(* CODESYS project CtaAppAntrieb_2.0.0.1.library
   Description: Antriebs Library der CTA
   Version: 2.0.0.1
   Title: CtaAppAntrieb
   Author: SIS
   DocFormat: reStructuredText
   LanguageModelAttribute: qualified-access-only
   Placeholder: CtaAppAntrieb
   DefaultNamespace: CtaAppAntrieb
   CompiledLibraryCompatibilityVersion: CODESYS V3.5 SP20 Patch 5
   Company: CTA

Project tree, tasks and I/O mapping:
  libraries: Standard, 3.5.18.0 (System); CtaAppBasic, 1.0.0.0 (CTA); CtaAppBmk, 2.0.0.0 (CTA); CtaSysConfig, 2.0.0.0 (CTA); VisuDialogs, 3.5.16.20 (System); VisuSymbols, 4.5.0.0 (System); CtaSysMotor, 1.0.0.0 (CTA); CtaAppReport, 2.0.0.0 (CTA); CtaVisHelp, 1.0.0.0 (CTA); CtaVisSymbols, 2.0.0.0 (CTA); CtaAppDumper, 2.0.0.0 (CTA); CtaAppInfluxLog, 1.0.0.1 (CTA); CtaSysIO, 2.0.0.0 (CTA); CtaAppModbusSpezifikation, 1.0.0.1 (CTA); CtaVisApps, 1.0.0.0 (CTA); CtaVisUser, 1.0.0.0 (CTA)
  40 Visualizations/
    ICON/
      ANTRIEB_RIGHT/
        ANTRIEB_RIGHT_BELOW/
          visualisation VIS_ANTRIEB_RIGHT_BELOW
          visualisation VIS_ANTRIEB_RigthBelowCheckIsEnabled
          visualisation VIS_ANTRIEB_RigthBelowCheckQuerry
        ANTRIEB_RIGHT_ABOVE/
          visualisation VIS_ANTRIEB_RigthAboveCheckQuerry
          visualisation VIS_ANTRIEB_RIGHT_ABOVE
          visualisation VIS_ANTRIEB_RigthAboveCheckIsEnabled
      ANTRIEB_BASE/
        visualisation CommandOn
        visualisation ValueUpDwn
        ICON/
          visualisation Icon_Left
          visualisation Icon_Right
        visualisation ValueDwnUp
      ANTRIEB_LEFT/
        ANTRIEB_LEFT_BELOW/
          visualisation VIS_ANTRIEB_LEFT_BELOW
          visualisation VIS_ANTRIEB_LeftBelowCheckIsEnabled
          visualisation VIS_ANTRIEB_LeftBelowCheckQuerry
        ANTRIEB_LEFT_ABOVE/
          visualisation VIS_ANTRIEB_LEFT_ABOVE
          visualisation VIS_ANTRIEB_LeftAboveCheckIsEnabled
          visualisation VIS_ANTRIEB_LeftAboveCheckQuerry
    POPUP/
      visualisation POPUP_ANTRIEB
      PARAMETER/
        visualisation VIS_ANTRIEB_PARAMETER
        visualisation VIS_ANTRIEB_PARAMETER_LISTE
        AT_ParameterBase/
          visualisation VIS_ANTRIEB_PARAMETER_BASE0
          visualisation VIS_ANTRIEB_PARAMETER_BASE
        AT_Data/
          visualisation VIS_ANTRIEB_PARAMETER_DATA0
          visualisation VIS_ANTRIEB_PARAMETER_DATA
        AT_Fuse/
          visualisation VIS_ANTRIEB_PARAMETER_FUSES0
          visualisation VIS_ANTRIEB_PARAMETER_FUSES
        AT_IO/
          visualisation VIS_ANTRIEB_PARAMETER_IO0
          visualisation VIS_ANTRIEB_PARAMETER_IO1
          visualisation VIS_ANTRIEB_PARAMETER_IO
          visualisation VIS_ANTRIEB_PARAMETER_IO2
          visualisation VIS_ANTRIEB_PARAMETER_IO3
          visualisation VIS_ANTRIEB_PARAMETER_IO4
        AT_InfluxDb/
          visualisation VIS_ANTRIEB_PARAMETER_TRENDLOG
          visualisation VIS_ANTRIEB_PARAMETER_TRENDLOG0
        visualisation VIS_ANTRIEB_POPUP_IO_ITF
      visualisation VIS_ANTRIEB_LISTE
      MANUAL/
        visualisation VIS_ANTRIEB_MANUAL
      OVERVIEW/
        visualisation VIS_ANTRIEB_OVERVIEW
      BUS/
        visualisation AT_BUS
        visualisation AT_BUS_SW0_Detail
        visualisation AT_BUS_CW0_Detail
        visualisation AT_BUS_CS
        visualisation AT_BUS_SW1_Detail
        visualisation AT_BUS_SW2_Detail
      REPORTS/
        visualisation VIS_ANTRIEB_REPORTS
      IO/
        visualisation VIS_ANTRIEB_IO0
        visualisation VIS_ANTRIEB_IO
        visualisation VIS_ANTRIEB_IO1
  30 Program Organization Units/
    function block fbAntrieb [ST]: proHandOn, proAuto, proHandOff, proHandOnY, proHardWareHandModulAktive, actConfig, proConfigError, proIconNr, P_scBase_fbrYMax, P_scBase_fbrYMin, P_scBase_fbtLeadTime, P_scBase_fbtRunAfterTime, P_scBase_fbxControllMb, P_scBase_fbxEnable, P_scBase_fbxRegulatet, P_scData_fbudiOperatingHours, P_scData_fbudiOperationStarts, P_scFuse_fbxDoesAlarm, P_scFuse_fbxEnable, P_scFuse_fbxInputMb, P_scInfluxDb_fbxEnable, P_scIO_IsHand_fbxEnable, P_scIO_IsHand_fbxInputMb, P_scIO_IsNoError_fbiMaxErrorRetryAllowed, P_scIO_IsNoError_fbiTypeOfAck, P_scIO_IsNoError_fbtDelayRun, P_scIO_IsNoError_fbtDelayStartSps, P_scIO_IsNoError_fbxDoesAlarm, P_scIO_IsNoError_fbxEnable, P_scIO_IsNoError_fbxInputMb, P_scIO_IsOn_fbiMaxErrorRetryAllowed, P_scIO_IsOn_fbiTypeOfAck, P_scIO_IsOn_fbtDelayRun, P_scIO_IsOn_fbtDelayStart, P_scIO_IsOn_fbxDoesAlarm, P_scIO_IsOn_fbxEnable, P_scIO_IsOn_fbxInputMb, P_scIO_IsReady_fbxEnable, P_scIO_IsReady_fbxInputMb, P_scIO_IsValue_fbiMaxErrorRetryAllowed, P_scIO_IsValue_fbiTypeOfAck, P_scIO_IsValue_fbrMaxDiff, P_scIO_IsValue_fbtDelayRun, P_scIO_IsValue_fbtDelayStart, P_scIO_IsValue_fbxDoesAlarm, P_scIO_IsValue_fbxEnable, P_scIO_IsValue_fbxInputMb, P_scIO_RevisionSwitch_fbxEnable, P_scIO_RevisionSwitch_fbxInputMb, P_scManual_fbrManualOnY, P_scManual_fbuiManualState, P_scManual_fbxAlowManualOn, P_scMotorFuse_fbxDoesAlarm, P_scMotorFuse_fbxEnable, P_scMotorFuse_fbxInputMb, proRefToRonYDumper, actMbControll, actMbState, proModbusTest, proModbusStateWord, proModbusControllWord, proIsOn, proIsError, proIsWarning, proIsRegulatet, proIsEnabled, actState, proMotorIsOn, proIsHandOnOrOff, proIsReady, proLeadTime, proRunAfterTime, proIsOnY, proLeadTimeAktive, proRunAfterTimeAktive, proRevisionSwitchOk, proCountedHours, proCountedStarts, proStateSymbol, proCountedError, proCountedInfo, proCountedWarning, proITF_REPORTMANAGER, proGetDI_IsOn, metDI_IsOn, proNotShowDI_IsOn, proIsOn_ITF, metDI_RevisionSwitchOk, proNotShowDI_RevisionSwitchOk, proGetDI_RevisionSwitchOK, proRevisionSwitch_ITF, metDI_NoError, proNotShowDI_NoError, proGetDI_NoError, proNoError_ITF, proGetDI_FuseOK, metDI_ITF_FuseOK, proNotShowDI_FuseOk, proFuse_ITF, metDI_ITF_MotorHand, proNotShowDI_MotorHand, proGetDI_MotorHand, proHandModul_ITF, metDI_IsReady, proNotShowDI_Ready, proGetDI_IsReady, proReady_ITF, metDI_MotorFuseOk, proNotShowDI_MotorFuseOk, proGetDI_MotorFuseOk, proMotorFuse_ITF, metDO_On, proOn_ITF, metAO_OnY, proOnY_ITF, proNotShowAI_ActualValue, metAI_ActualValue, proGetAI_ActualValue, proActualValue_ITF, proOnY, proOn, actVorlaufNachlauf, actPrioOfControll, actResetOnDisable, proEn, proEnSymbol, actTrendLog, actReport, proLockDown, proAvailable, proAcknowlege
    function fcGetBigerStringValue [ST]
    function fcCheckQuerryAndIconReturn [ST]
  00000000-0000-0000-0000-000000000000|D:\CoDeSys\LibrariesV3\trunk\Intern\CAA\CAA Template\3.4.0.0 draft\Placeholder.xml
  00000000-0000-0000-0000-000000000000|D:\CoDeSys\LibrariesV3\trunk\Intern\CAA\CAA Template\3.2.0.3 draft\Prefix.pdf
  00000000-0000-0000-0000-000000000000|D:\CoDeSys\LibrariesV3\trunk\Intern\CAA\CAA Template\3.5.2.0 draft\Placeholder.xml
  20 Structs/
    data type scParameter
    IO/
      data type scIO_IsOn
      data type scIO_IsNoError
      data type scIO_IsReady
      data type scIO_RevisionSwitch
      data type scIO_IsValue
      data type scIO_IsHand
    BASE/
      data type scBase
    DATA/
      data type scData
    FUSE/
      data type scFuse
      data type scMotorFuse
    InfluxDb/
      data type scInfluxDb
    MANUAL/
      data type scManual
  50 Images/
  10 Documenation/
    global variables VersionHistory
    global variables readMe
  21 Interface/
    interface ITF_ANTRIEB: proModbusTest, proModbusStateWord, proModbusControllWord, proConfigError, P_scIO_IsHand_fbxEnable, P_scIO_IsHand_fbxInputMb, P_scIO_IsNoError_fbxEnable, P_scIO_IsNoError_fbxInputMb, P_scIO_IsNoError_fbxDoesAlarm, P_scIO_IsNoError_fbtDelayStartSps, P_scIO_IsNoError_fbtDelayRun, P_scIO_IsNoError_fbiTypeOfAck, P_scIO_IsNoError_fbiMaxErrorRetryAllowed, P_scIO_IsOn_fbxInputMb, P_scIO_IsOn_fbxEnable, P_scIO_IsOn_fbtDelayStart, P_scIO_IsOn_fbxDoesAlarm, P_scIO_IsOn_fbtDelayRun, P_scIO_IsOn_fbiTypeOfAck, P_scIO_IsOn_fbiMaxErrorRetryAllowed, P_scIO_IsReady_fbxEnable, P_scIO_IsReady_fbxInputMb, P_scIO_IsValue_fbxInputMb, P_scIO_IsValue_fbxEnable, P_scIO_IsValue_fbxDoesAlarm, P_scIO_IsValue_fbtDelayStart, P_scIO_IsValue_fbtDelayRun, P_scIO_IsValue_fbiTypeOfAck, P_scIO_IsValue_fbiMaxErrorRetryAllowed, P_scIO_IsValue_fbrMaxDiff, P_scIO_RevisionSwitch_fbxEnable, P_scIO_RevisionSwitch_fbxInputMb, P_scBase_fbxEnable, P_scBase_fbxRegulatet, P_scBase_fbxControllMb, P_scBase_fbrYMin, P_scBase_fbrYMax, P_scBase_fbtLeadTime, P_scBase_fbtRunAfterTime, P_scFuse_fbxEnable, P_scFuse_fbxInputMb, P_scFuse_fbxDoesAlarm, P_scMotorFuse_fbxInputMb, P_scMotorFuse_fbxEnable, P_scMotorFuse_fbxDoesAlarm, P_scManual_fbxAlowManualOn, P_scManual_fbuiManualState, P_scManual_fbrManualOnY, P_scInfluxDb_fbxEnable, P_scData_fbudiOperationStarts, P_scData_fbudiOperatingHours, proRefToRonYDumper, proCountedError, proCountedInfo, proITF_REPORTMANAGER, proCountedWarning, proCountedHours, proCountedStarts, proGetDI_MotorHand, proNotShowDI_MotorHand, proHandModul_ITF, proNotShowAI_ActualValue, proGetAI_ActualValue, proActualValue_ITF, proNotShowDI_NoError, proGetDI_NoError, proNoError_ITF, proNotShowDI_RevisionSwitchOk, proGetDI_RevisionSwitchOK, proRevisionSwitch_ITF, proNotShowDI_IsOn, proGetDI_IsOn, proIsOn_ITF, proNotShowDI_MotorFuseOk, proGetDI_MotorFuseOk, proMotorFuse_ITF, proNotShowDI_FuseOk, proGetDI_FuseOK, proFuse_ITF, proNotShowDI_Ready, proGetDI_IsReady, proReady_ITF, proOn_ITF, proOnY_ITF, proIsRegulatet, proIsHandOnOrOff, proRunAfterTimeAktive, proLeadTimeAktive, proIsReady, proAuto, proHandOn, proIsError, proIsWarning, proEn, proHardWareHandModulAktive, proIsEnabled, proMotorIsOn, proHandOff, proRevisionSwitchOk, proHandOnY, proEnSymbol, proIsOn, proIsOnY, proLeadTime, proOn, proOnY, proRunAfterTime, proStateSymbol, proLockDown, proAvailable, proAcknowlege, proIconNr
  11 Library Parameter/
  12 Konstanten/
    global variables GlobalKonstant
  60 Textlisten/
    text list GlobalTextList
    text list Error
    text list Info
    text list Warnung
  13 Globale Variablen/
  5ce3da45-db07-42e7-a21c-a00fff4ed8f6|C:\Users\sis\Downloads\dip-switch.svg
  5ce3da45-db07-42e7-a21c-a00fff4ed8f6|C:\Users\sis\Downloads\lightning-bolt-circle.svg
  5ce3da45-db07-42e7-a21c-a00fff4ed8f6|C:\Users\sis\Downloads\sine-wave.svg
  5ce3da45-db07-42e7-a21c-a00fff4ed8f6|C:\Users\sis\Downloads\eye.svg
  5ce3da45-db07-42e7-a21c-a00fff4ed8f6|C:\Users\sis\Downloads\lan.svg
*)

// 20 Structs/scParameter
{attribute 'pack_mode' := '1'} 
TYPE scParameter :
    STRUCT
		
        scBase              :   scBase;					// Basisparameter		
        scFuse              :   scFuse;					// Parameter Sicherung
        scMotorFuse         :   scMotorFuse;			// Parameter Motorsicherung
        scIO_RevisionSwitch :   scIO_RevisionSwitch;	// Parameter Revisionsschalter 
        scIO_IsReady        :   scIO_IsReady;   		// Parameter Bereitmeldung
        scIO_IsOn           :   scIO_IsOn;				// Parameter Betriebsrückmeldung
        scIO_IsNoError      :   scIO_IsNoError;			// Parameter Störmeldung
        scIO_IsValue        :   scIO_IsValue;			// Parameter Istwert
        scIO_IsHand         :   scIO_IsHand;        	// Parameter Handwert
        scManual            :   scManual;				// Parameter Handbedienung
        scData              :   scData;					// Parameter Betriebsdaten 
        scInfluxDb          :   scInfluxDb;				// Parameter Datenbankaufzeichung
    END_STRUCT
END_TYPE

// 20 Structs/IO/scIO_IsOn
{attribute 'pack_mode' := '1'} 
TYPE scIO_IsOn :
    STRUCT
        fbxEnable                    : CtaSysConfig.fbBOOL;	// Betriebsrückmeldung wird ausgewertet
        fbxInputMb                   : CtaSysConfig.fbBOOL; // Betriebsrückmeldung via Modbus  
        fbxDoesAlarm                 : CtaSysConfig.fbBOOL; // Ausstehende Betriebsrückmeldung löst Fehler aus 
        fbtDelayStart                : CtaSysConfig.fbTIME; // Verzögerung für Srörungsausgabe
        fbtDelayRun                  : CtaSysConfig.fbTIME; // Verzögerung für Störungsausgabe während Betrieb 
        fbiTypeOfAck               	 : CtaSysConfig.fbINT;  // Art der FehlerQuittierung 0 = Automatisch, 1 = Quittierpflichtig, 2 = Selbstquittierend bis N  
        fbiMaxErrorRetryAllowed      : CtaSysConfig.fbINT;  // Anzahl möglicher Selbstquittierungen    
    END_STRUCT
END_TYPE

// 20 Structs/IO/scIO_IsNoError
{attribute 'pack_mode' := '1'} 
TYPE scIO_IsNoError :
    STRUCT
        fbxEnable                    : CtaSysConfig.fbBOOL;	// Störkontakt wird ausgewertet
        fbxInputMb                   : CtaSysConfig.fbBOOL; // Störkontaktstatus via Modbus
        fbxDoesAlarm                 : CtaSysConfig.fbBOOL;	// Störung löst Fehler aus
        fbtDelayStartSps             : CtaSysConfig.fbTIME; // Verzögerung für Srörungsausgabe
        fbtDelayRun                  : CtaSysConfig.fbTIME; // Verzögerung für Störungsausgabe während Betrieb 
        fbiTypeOfAck               	 : CtaSysConfig.fbINT;	// Art der FehlerQuittierung 0 = Automatisch, 1 = Quittierpflichtig, 2 = Selbstquittierend bis N 
        fbiMaxErrorRetryAllowed      : CtaSysConfig.fbINT;	// Anzahl möglicher Selbstquittierungen
    END_STRUCT
END_TYPE

// 20 Structs/IO/scIO_IsReady
{attribute 'pack_mode' := '1'} 
TYPE scIO_IsReady :
    STRUCT
        fbxEnable                    : CtaSysConfig.fbBOOL;	// Bereitmeldung wird ausgewertet 
        fbxInputMb                   : CtaSysConfig.fbBOOL; // Bereitmeldung üver Modbus         
    END_STRUCT
END_TYPE

// 20 Structs/IO/scIO_RevisionSwitch
{attribute 'pack_mode' := '1'} 
TYPE scIO_RevisionSwitch :
    STRUCT
        fbxEnable                   : CtaSysConfig.fbBOOL;	// Revisionsschalter wird ausgewertet
        fbxInputMb                  : CtaSysConfig.fbBOOL;	// Revisionsschalterstatus via Modbus
    END_STRUCT
END_TYPE

// 20 Structs/IO/scIO_IsValue
{attribute 'pack_mode' := '1'} 
TYPE scIO_IsValue :
    STRUCT
        fbxEnable                    : CtaSysConfig.fbBOOL;	// Iststellwert wird ausgewertet
        fbxInputMb                   : CtaSysConfig.fbBOOL; // Iststellwert via Modbus    
        fbxDoesAlarm                 : CtaSysConfig.fbBOOL; // Zugrosse Abweichung löst Fehler aus  
        fbrMaxDiff                   : CtaSysConfig.fbREAL; // Maximal zulässige abweichung von Soll- zu Iststellwert
        fbtDelayStart                : CtaSysConfig.fbTIME; // Verzögerung für Srörungsausgabe
        fbtDelayRun                  : CtaSysConfig.fbTIME; // Verzögerung für Störungsausgabe während Betrieb 
		fbiTypeOfAck				 : CtaSysConfig.fbINT;  // Art der FehlerQuittierung 0 = Automatisch, 1 = Quittierpflichtig, 2 = Selbstquittierend bis N  
		fbiMaxErrorRetryAllowed		 : CtaSysConfig.fbINT;  // Anzahl möglicher Selbstquittierungen            
    END_STRUCT
END_TYPE

// 20 Structs/IO/scIO_IsHand
{attribute 'pack_mode' := '1'} 
TYPE scIO_IsHand :
    STRUCT
        fbxEnable                   : CtaSysConfig.fbBOOL;	// Handmodul wird ausgewertet
        fbxInputMb                  : CtaSysConfig.fbBOOL;	// Handmodulstatus via Modbus
    END_STRUCT
END_TYPE

// 20 Structs/BASE/scBase
{attribute 'pack_mode' := '1'} 
TYPE scBase :
    STRUCT
        fbxEnable       :   CtaSysConfig.fbBOOL;	// Antriebsbaustein wird abgearbeitet
        fbxRegulatet    :   CtaSysConfig.fbBOOL;	// Antriebsstellwert wird geregelt
        fbxControllMb   :   CtaSysConfig.fbBOOL;	// Antriebsansteuerung erfolgt über Modbus
        fbrYMin         :   CtaSysConfig.fbREAL;	// Minimalstellwert des Antriebes
        fbrYMax         :   CtaSysConfig.fbREAL;	// Maximalstellwert des Antriebes
        fbtLeadTime     :   CtaSysConfig.fbTIME;	// Vorlaufzeit des Antriebs
        fbtRunAfterTime :   CtaSysConfig.fbTIME;	// Nachlaufzeit des Antriebs
    END_STRUCT
END_TYPE

// 20 Structs/DATA/scData
{attribute 'pack_mode' := '1'} 
TYPE scData :
    STRUCT
        fbudiOperationStarts    :   CtaSysConfig.fbUDINT;	// Anzahl Einschaltungen des Antriebs
        fbudiOperatingHours     :   CtaSysConfig.fbUDINT;	// Anzahl Betriebsstunden des Antriebs
    END_STRUCT
END_TYPE

// 20 Structs/FUSE/scFuse
{attribute 'pack_mode' := '1'} 
TYPE scFuse :
    STRUCT
        fbxEnable               : CtaSysConfig.fbBOOL;	// Sicherung ist vorhanden
        fbxInputMb              : CtaSysConfig.fbBOOL;	// Sicherungsstatus via Modbus
        fbxDoesAlarm            : CtaSysConfig.fbBOOL;	// Defekte Sicherung löst Fehler aus
    END_STRUCT
END_TYPE

// 20 Structs/FUSE/scMotorFuse
{attribute 'pack_mode' := '1'} 
TYPE scMotorFuse :
    STRUCT
        fbxEnable             : CtaSysConfig.fbBOOL;	// Sicherung ist vorhanden
        fbxInputMb            : CtaSysConfig.fbBOOL;    // Sicherungsstatus via Modbus
        fbxDoesAlarm          : CtaSysConfig.fbBOOL;    // Defekte Sicherung löst Fehler aus  
    END_STRUCT
END_TYPE

// 20 Structs/InfluxDb/scInfluxDb
{attribute 'pack_mode' := '1'} 
TYPE scInfluxDb :
    STRUCT
        fbxEnable       :   CtaSysConfig.fbBOOL;	// Aktivierung der Trendaufzeichnung
    END_STRUCT
END_TYPE

// 20 Structs/MANUAL/scManual
{attribute 'pack_mode' := '1'} 
TYPE scManual :
    STRUCT
        fbxAlowManualOn         : CtaSysConfig.fbBOOL; 	// Manuelle ansteuerung des Antriebs zulässig   
        fbuiManualState         : CtaSysConfig.fbUINT;	// 0 = Auto ; 1 = Manual Off 2 = Manual On
        fbrManualOnY            : CtaSysConfig.fbREAL; 	// Manueller Stellwert für Antrieb
    END_STRUCT
END_TYPE

// 10 Documenation/VersionHistory
(* 

.. image:: ../../Images/CTA_Logo.jpg
   :align: right
   :width: 15% 

**Vorlage**   


============ =========== =========== ============================================
**Date**     **Version** **Author**  **Change**
------------ ----------- ----------- --------------------------------------------
04.03.2021   0.0.0.0     SIS         Vorlage erstellt

============ =========== =========== ============================================


*)
VAR_GLOBAL
    stInfo : STRING:= '0.0.0.0, Vorlage, CTA';
END_VAR

// 10 Documenation/readMe

(*

**ReadMe**
 
|	**Empfehlung**
|
|	Die Bibliothek CtaAppAntrieb wurde universal gestaltet, dadurch können verschiedene Komponenten damit angesteuert werden.
|	Instanzieren Sie den CtaAppAntrieb.fbAntrieb in ihrem Funktionsbaustein oder POU beispielsweise als fbPumpeX oder fbVentiX abhängig der Komponente. (X = Nr.) 
|	Deklarieren Sie die Struktur Variable welche als Parameter und zur ansteuerung dienen wie im Code beispiel.
|  
| *Beispiel* 

+-----------------------+---------------------------------------------------------------------------------------------------------------------------------------------------------------------------------------------------------------------------------------------------------------------------------------------------------------------------------------------------------------------------------------------------------------------------------------+
| Beschreibung          |  Code                                                                                                                                                                                                                                                                                                                                                                                                                                 |
+=======================+=======================================================================================================================================================================================================================================================================================================================================================================================================================================+
| Pou oder SmFb         | .. code-block:: codesys                                                                                                                                                                                                                                                                                                                                                                                                               |
|                       |                                                                                                                                                                                                                                                                                                                                                                                                                                       |
|                       |	// Deklaration als VAR im POU oder dem selbsterstellten Funktionsbaustein                                                                                                                                                                                                                                                                                                                                                       	|
|                       |   VAR   																																																																																																								|
|						|	    (*Pumpe1*)																																																		 																																																				|
|						|		fbPumpe1			: CtaAppAntrieb.fbAntrieb;                                                                                                                                                                                                                                                                                                                                                              					|
|                       | 		(*Ventilator1*)																																																																																																					|
| 						|		fbVenti1			: CtaAppAntrieb.fbAntrieb;																																																																																													|
| 						|	END_VAR                                                                                                                                                                                                                                                                                                                                                                                                                         	|
+-----------------------+---------------------------------------------------------------------------------------------------------------------------------------------------------------------------------------------------------------------------------------------------------------------------------------------------------------------------------------------------------------------------------------------------------------------------------------+
| Code für Init         | .. code-block:: codesys                                                                                                                                                                                                                                                                                                                                                                                                               |
|                       |   																																																																																																									|
| 						|	// Kopieren des nachfolgenden Codes in eine Action zur Initialisierung der Parameter. Zum Beispiel actConfig.																																																																														|
|                       |	{region "Parameter Pumpe1"}                                                                                                                                                                                                                                                                                                                                                                                                     	|
| 						|		(*Basis*)																																																																																																						|
|						|		fbPumpe1.scParameter.scBase.fbxEnable               		(_wertInit :=  TRUE																			);		//P1 Ein- Ausschalten des Antriebs																																																								|
|						|		fbPumpe1.scParameter.scBase.fbxRegulatet					(_wertInit :=  TRUE																			);		//P2 Antrieb ist geregelt / nicht geregelt																																																						| 
|						|		fbPumpe1.scParameter.scBase.fbxControllMb					(_wertInit := FALSE																			);		//P3 Ansteuerung oder Signalauswertung über Modbus																																																				| 
|						|		fbPumpe1.scParameter.scBase.fbrYMin							(_wertInit :=   0.0									, _minInit :=   0.0, _maxInit := 100.0	);		//P4 Minimaler Stellwert des Antriebs																																																							| 
|						|		fbPumpe1.scParameter.scBase.fbrYMax							(_wertInit := 100.0									, _minInit :=   0.0, _maxInit := 100.0	);		//P5 Maximaler Stellwert des Antriebs																																																							|
|						|		fbPumpe1.scParameter.scBase.fbtLeadTime						(_wertInit := T#30S									, _minInit :=      , _maxInit :=		);		//P6 Vorlaufzeit des Antriebs																																																									| 
|						|		fbPumpe1.scParameter.scBase.fbtRunAfterTime					(_wertInit := T#60S									, _minInit :=	   , _maxinit :=		);		//P7 Nachlaufzeit des Antriebs																																																									| 
|						|		(*Sicherungen*)																																																		 																																																			| 
|						|		fbPumpe1.scParameter.scFuse.fbxEnable						(_wertInit := FALSE																			);		//P8 Sicherung ist vorhanden / nicht vorhanden																	    																																			| 
|						|		fbPumpe1.scParameter.scFuse.fbxInputMb						(_wertInit := FALSE																			);		//P9 Ansteuerung oder Signalauswertung über Modbus																												    																							| 
|						|		fbPumpe1.scParameter.scFuse.fbxDoesAlarm					(_wertInit := FALSE																			);		//P10 Abfallendes Signal löst Fehler aus																											    																										| 
|						|		(*Motorsicherung*)																																																											 																																	  								| 
|						|		fbPumpe1.scParameter.scMotorFuse.fbxEnable					(_wertInit := FALSE																			);		//P11 Leistungsschutzschalter ist vorhanden / nicht vorhanden																    																																| 
|						|		fbPumpe1.scParameter.scMotorFuse.fbxInputMb					(_wertInit := FALSE																			);		//P12 Ansteuerung oder Signalauswertung über Modbus																																								   	 											| 
|						|		fbPumpe1.scParameter.scMotorFuse.fbxDoesAlarm				(_wertInit := FALSE																			);		//P13 Abfallendes Signal löst Fehler aus																														    																							| 
|						|		(*Revisionsschalter*)																																																											 																																							    | 
|						|		fbPumpe1.scParameter.scIO_RevisionSwitch.fbxEnable			(_wertInit := FALSE																			);		//P14 Revisionsschalter ist vorhanden / nicht vorhanden																																				    														| 
|						|		fbPumpe1.scParameter.scIO_RevisionSwitch.fbxInputMb			(_wertInit := FALSE																			);		//P15 Ansteuerung oder Signalauswertung über Modbus																																		    																	| 
|						|		(*Ready- Input*)																																																																																																			    | 
|						|		fbPumpe1.scParameter.scIO_IsReady.fbxEnable					(_wertInit := FALSE																			);		//P16 Readysignal ist vorhanden / nicht vorhanden																																	    																		| 
|						|		fbPumpe1.scParameter.scIO_IsReady.fbxInputMb				(_wertInit := FALSE																			);		//P17 Ansteuerung oder Signalauswertung über Modbus																																										    									| 
|						|		(*Betriebsrückmeldung*)																																																										 																																								    | 
|						|		fbPumpe1.scParameter.scIO_IsOn.fbxEnable					(_wertInit := FALSE																			);		//P18 Betriebsrückmeldung ist vorhanden / nicht vorhanden																														   																				| 
|						|		fbPumpe1.scParameter.scIO_IsOn.fbxInputMb					(_wertInit := FALSE																			);		//P19 Ansteuerung oder Signalauswertung über Modbus																																								    											| 
|						|		fbPumpe1.scParameter.scIO_IsOn.fbxDoesAlarm					(_wertInit := FALSE																			);		//P20 Fehlendes oder abfallendes Signal löst Fehler aus				   																																															| 
|						|		fbPumpe1.scParameter.scIO_IsOn.fbtDelayStart				(_wertInit := T#00S									, _minInit :=      , _maxInit :=  		);		//P21 Verzögerung der Fehlerausgabe nach Start																						   																															| 
|						|		fbPumpe1.scParameter.scIO_IsOn.fbtDelayRun					(_wertInit := T#00S									, _minInit :=      , _maxInit :=  		);		//P22 Verzögerung der Fehlerausgabe während Betrieb															    																																				| 
|						|		fbPumpe1.scParameter.scIO_IsOn.fbiTypeOfAck					(_wertInit :=     1									, _minInit :=     0, _maxInit :=    2	);		//P23 Art der Quittierung des Fehlers (auto, quittierend, quittierend bid n Meldung																																												|
|						|		fbPumpe1.scParameter.scIO_IsOn.fbiMaxErrorRetryAllowed		(_wertInit :=     3									, _minInit :=     0, _maxInit :=    5	);		//P24 Maximale Anzahl Wiederholungen bis zur Sperrung der Anlage																																																|
|						|		(*Fehler- Input*)																																																																																																			    | 
|						|		fbPumpe1.scParameter.scIO_IsNoError.fbxEnable				(_wertInit := FALSE																			);		//P25 Fehlerinput ist vorhanden / nicht vorhanden																																		    																	| 
|						|		fbPumpe1.scParameter.scIO_IsNoError.fbxInputMb				(_wertInit := FALSE																			);		//P26 Ansteuerung oder Signalauswertung über Modbus																																																			    | 
|						|		fbPumpe1.scParameter.scIO_IsNoError.fbxDoesAlarm			(_wertInit := FALSE																			);		//P27 Fehlendes oder abfallendes Signal löst Fehler aus				   																																														    | 
|						|		fbPumpe1.scParameter.scIO_IsNoError.fbtDelayStartSps		(_wertInit := T#00S									, _minInit :=      , _maxInit :=  		);		//P28 Verzögerung der Fehlerausgabe nach Start																																																			    	| 
|						|		fbPumpe1.scParameter.scIO_IsNoError.fbtDelayRun				(_wertInit := T#00S									, _minInit :=      , _maxInit :=  		);		//P29 Verzögerung der Fehlerausgabe während Betrieb																																																			    | 
|						|		fbPumpe1.scParameter.scIO_IsNoError.fbiTypeOfAck			(_wertInit :=     1 								, _minInit :=     0, _maxInit :=    2	);		//P30 Art der Quittierung des Fehlers (auto, quittierend, quittierend bid n Meldung																																										    	| 
|						|		fbPumpe1.scParameter.scIO_IsNoError.fbiMaxErrorRetryAllowed	(_wertInit :=     3 								, _minInit :=     0, _maxInit :=    5	);		//P31 Maximale Anzahl Wiederholungen bis zur Sperrung der Anlage																																										    					| 
|						|		(*Ist - Wert*)																																																																																																				    | 
|						|		fbPumpe1.scParameter.scIO_IsValue.fbxEnable					(_wertInit := FALSE																			);		//P32 Rückmeldung des Istwerts ist vorhanden / nicht vorhanden																																																	| 
|						|		fbPumpe1.scParameter.scIO_IsValue.fbxInputMb				(_wertInit := FALSE																			);		//P33 Ansteuerung oder Signalauswertung über Modbus																																																				| 
|						|		fbPumpe1.scParameter.scIO_IsValue.fbxDoesAlarm				(_wertInit := FALSE																			);		//P34 Unter oder überschreitung der Maximal erlaubten Differenz löst Fehler aus				   																																									| 
|						|		fbPumpe1.scParameter.scIO_IsValue.fbrMaxDiff				(_wertInit :=   0.0									, _minInit :=      , _maxInit :=		);		//P34 Maximal erlaubte Differenz des Stell- zum Istwert  			   																																															| 
|						|		fbPumpe1.scParameter.scIO_IsValue.fbtDelayStart				(_wertInit := T#00S									, _minInit :=      , _maxInit :=    	);		//P36 Verzögerung der Fehlerausgabe nach Start																																																					| 
|						|		fbPumpe1.scParameter.scIO_IsValue.fbtDelayRun				(_wertInit := T#00S									, _minInit :=      , _maxInit :=    	);		//P37 Verzögerung der Fehlerausgabe während Betrieb																																																				| 
|						|		fbPumpe1.scParameter.scIO_IsValue.fbiTypeOfAck				(_wertInit :=     1									, _minInit :=     0, _maxInit :=    2	);		//P38 Art der Quittierung des Fehlers (auto, quittierend, quittierend bid n Meldung																																												| 
|						|		fbPumpe1.scParameter.scIO_IsValue.fbiMaxErrorRetryAllowed 	(_wertInit :=     3									, _minInit :=     0, _maxInit :=    5	);		//P39 Maximale Anzahl Wiederholungen bis zur Sperrung der Anlage																																																| 
|						|		(*Sollwertdämpfung*)																																																																																																			|
|						|		fbPumpe1.fbDumperRonY.scParameter.fbrTup					(_wertInit :=   1.0                                 , _minInit :=       , _maxInit :=    	);      //P34 Maximal erlaubte Differenz des Stell- zum Istwert																																																			|
|						|		fbPumpe1.fbDumperRonY.scParameter.fbrTdown					(_wertInit :=   1.0                                 , _minInit :=       , _maxInit :=    	);      //P34 Maximal erlaubte Differenz des Stell- zum Istwert																																																			|
|						|		fbPumpe1.fbDumperRonY.scParameter.fbrBand					(_wertInit := 100.0                                 , _minInit :=       , _maxInit :=    	);      //P34 Maximal erlaubte Differenz des Stell- zum Istwert																																																			|
|						|		fbPumpe1.fbDumperRonY.scParameter.fbxInExpOut				(_wertInit := FALSE                                                                      	);      //P42 Handansteuerung zulassen / nicht zulassen																																																					|
|						|		(*Handmodul*)																																																		 																																																		    | 
|						|		fbPumpe1.scParameter.scIO_IsHand.fbxEnable					(_wertInit := FALSE																			);		//P40 Handmodul ist vorhanden / nicht vorhanden																																																					| 
|						|		fbPumpe1.scParameter.scIO_IsHand.fbxInputMb					(_wertInit := FALSE																			);		//P41 Ansteuerung oder Signalauswertung über Modbus																																																				| 
|						|		(*Manuelle Ansteuerung*)																																																																																																	    | 
|						|		fbPumpe1.scParameter.scManual.fbxAlowManualOn				(_wertInit :=  TRUE																			);		//P42 Handansteuerung zulassen / nicht zulassen																																																					| 
|						|		fbPumpe1.scParameter.scManual.fbuiManualState				(_wertInit := 	  0									, _minInit :=     0, _maxInit :=    2	);		//P43 Ansteuerungsmodus des Ventils (auto, manuell, gesperrt)																																																	| 
|						|		fbPumpe1.scParameter.scManual.fbrManualOnY					(_wertInit := 	  0									, _minInit :=     0, _maxInit :=  100	);		//P44 Manueller Stellwert für den Antrieb																																																						| 
|						|		(*Betriebsdaten*)																																																																																																			    | 
|						|		fbPumpe1.scParameter.scData.fbudiOperationStarts			(_wertInit := 	  0									, _minInit :=     0, _maxInit :=    0	);		//P45 Betriebsstarts der Anlage																																																									| 
|						|		fbPumpe1.scParameter.scData.fbudiOperatingHours				(_wertInit :=     0									, _minInit :=     0, _maxInit :=    0	);		//P46 Betriebsstunden der Anlage																																																								| 
|						|		(*Trendlog*)																																																																																																					| 
|						|		fbPumpe1.scParameter.scInfluxDb.fbxEnable					(_wertInit :=  TRUE																			);		//P47 Aktiverung / Deaktivierung der Trenddaten 																																																				| 
|						|	{endregion}                                                                                                                                                      																																																																	| 
+-----------------------+---------------------------------------------------------------------------------------------------------------------------------------------------------------------------------------------------------------------------------------------------------------------------------------------------------------------------------------------------------------------------------------------------------------------------------------+
*)                                                                                                                                                                                                                                                                                                                                                                                                                                                               
 VAR_GLOBAL                                                                                                                                                                                                                                                                                                                                                                                                                                                      
    xReadMeDone              :   BOOL;                                                                                                                                                                                                                                                                                                                                                                                                                           
END_VAR

// 12 Konstanten/GlobalKonstant
{attribute 'qualified_only'}
VAR_GLOBAL CONSTANT 	
	stReportTextListError   : CtaAppReport.stReportTextList := 'CtaAppAntrieb.Error';	// Textlistenbezeichnung für Fehler
	stReportTextListWarning : CtaAppReport.stReportTextList := 'CtaAppAntrieb.Warnung';	// Textlistenbezeichnung für Warnungen
	stReportTextListInfo    : CtaAppReport.stReportTextList := 'CtaAppAntrieb.Info';	// Textlistenbezeichnung für Informationen 
    uiMaxParameter          : UINT := 47;												// Maximale Anzahl Parameter pro Antrieb
END_VAR

// 30 Program Organization Units/fbAntrieb
FUNCTION_BLOCK fbAntrieb EXTENDS CtaAppBmk.fbBMK IMPLEMENTS ITF_ANTRIEB 
VAR_INPUT
    xRelease                    :   BOOL;
    rRelease                    :   REAL;
    xSafetyStop                 :   BOOL;
END_VAR                         
VAR_OUTPUT                      
    (* Commmands *)               
    xOn                         :   BOOL; 
    rOnY                        :   REAL;
    (* State Out*)              
    xIsOn                       :   BOOL;
END_VAR                 
VAR                     
    (* State Intern*)      
    scEWI                       :   CtaAppReport.scReportNr;                 
    xIsWarning                  :   BOOL;
    _xIsWarning                 :   BOOL;
    xIsError                    :   BOOL;
    _xIsError                   :   BOOL;
    xIsRegulatet                :   BOOL;
    xIsEnabled                  :   BOOL;
    xIsHand                     :   BOOL;
    xIsHandOn                   :   BOOL;
    xIsHandOff                  :   BOOL;
    xIsAuto                     :   BOOL;   
    xConfigError                :   BOOL;
	uiIconNr					:	UINT;
	fbDumperRonY				:	CtaAppDumper.fbDumper;
	(* ITF OUT*)
	ITF_xOn						:	CtaSysIO.ITF_IO;
	ITF_rOnY					:	CtaSysIO.ITF_IO;
    (* Inputs *)
	// Fuse
    xFuseOk                     :   BOOL;
    xInFuseOk                   :   BOOL;
    xInFuseOkMb                 :   BOOL;
	ITF_Fuse					:	CtaSysIO.ITF_IO;
	// Motor fuse
    xMotorFuseOk                :   BOOL;    
    xInMotorFuseOk              :   BOOL;
    xInMotorFuseOkMb            :   BOOL;
	ITF_MotorFuse				:	CtaSysIO.ITF_IO;
	// No Error
    xMotorNoError               :   BOOL;   
    xInMotorNoError             :   BOOL;
    xInMotorNoErrorMb           :   BOOL;
	ITF_MotorNoError			:	CtaSysIO.ITF_IO;
	// Is ready
    xMotorIsReady               :   BOOL;
    xInMotorIsReady             :   BOOL;
    xInMotorIsReadyMb           :   BOOL;
	ITF_MotorIsReady			:	CtaSysIO.ITF_IO;
	// Is on
    xMotorIsOn                  :   BOOL;
    xInMotorIsOn                :   BOOL;
    xInMotorIsOnMb              :   BOOL;
	ITF_MotorIsOn				:	CtaSysIO.ITF_IO;
	// Revision switch
    xMotorRevisionSwitchOff     :   BOOL;
    xMotorRevisionSwitchOn      :   BOOL;
    xInMotorRevisionSwitchOn    :   BOOL;   
    xInMotorRevisionSwitchOnMb  :   BOOL;
	ITF_RevisionSwitch			:	CtaSysIO.ITF_IO;
	// Motor Hand 
    xMotorHand                  :   BOOL;
    xInMotorHand                :   BOOL;
    xInMotorHandMb              :   BOOL;
	ITF_MotorHand				:	CtaSysIO.ITF_IO;
	// Actual Value
    rInActualValue              :   REAL; 
	ITF_ActualValue				:	CtaSysIO.ITF_IO;
    (* Motor *)
    xReleaseFromModBus          :   BOOL;
    xReleaseControllPrio        :   BOOL;
    rReleaseFromModBus          :   REAL;
    rReleaseControllPrio        :   REAL;
    xReleaseMotor               :   BOOL;
    rReleaseScaled              :   REAL;
    xErrorIsOn                  :   BOOL;
    xErrorMotorError            :   BOOL;    
    xSafetyStopMotor            :   BOOL;    
    TON_LeadTime                :   TON;
    TOF_RunAfter                :   TOF;
    tLeadTime				    :	TIME;                                   // Aktuelle Nachlaufzeit 
    xLeadTimeAktive             :   BOOL;
    tRunAfter					:	TIME;                                   // Aktuelle Vorlaufzeit          
    xRunAfterAktive             :   BOOL;    
    fbMotor                     :   CtaSysMotor.fbMotor;
    fbCheckMotorIsOn            :   CtaSysMotor.fbSafetyInput;    
    fbCheckIsError              :   CtaSysMotor.fbSafetyInput; 
    fbDataCount                 :	CtaSysMotor.fbOperationDataCounter;          
    (* Modbus *)
    xModbusTest                 :   BOOL;
    ayMbControllWord            :   ARRAY[0..3] OF WORD;
    ayMbStateWord               :   ARRAY[0..3] OF WORD;
    (* Parameter *)
    fbConfigFile                :   CtaSysConfig.fbConfigFile;
    scParameter                 :   scParameter;
    (* Reports *)	
    fbReportManager			    :   CtaAppReport.fbReportManager;      
    difor					    :	DINT;                                                                    
    ayErrorReporter				:	ARRAY[1..5] OF CtaAppReport.fbReporter;
	ayWarningReporter			:	ARRAY[1..5] OF CtaAppReport.fbReporter;
	(* Trendlogs *)
	fbTrendxOn					:	CtaAppInfluxLog.FB_LOG_NODE_BOOL;
	fbTrendxIsOn				:	CtaAppInfluxLog.FB_LOG_NODE_BOOL;
	fbTrendxMotorIsOn			:	CtaAppInfluxLog.FB_LOG_NODE_BOOL;
	fbTrendrOnY					:	CtaAppInfluxLog.FB_LOG_NODE_REAL;
	fbTrendrIsOnY				:	CtaAppInfluxLog.FB_LOG_NODE_REAL;
	fbTrendxError				:	CtaAppInfluxLog.FB_LOG_NODE_BOOL;
    (* Collector *)
    diArrayPosition             :   DINT;
END_VAR

(* Config *)
actConfig();

(* Motor Command *)
IF xIsEnabled AND NOT xConfigError THEN
    (* Modbus Controll *)
    actMbControll();
    (* Controll Prio *)
    actPrioOfControll();	
    (* Ckeck motorfeedback if *)       
    IF scParameter.scIO_IsOn.fbxDoesAlarm.proValue > scParameter.scIO_IsOn.fbxEnable.proValue THEN
        // Alarm Only if Enabled
        scParameter.scIO_IsOn.fbxDoesAlarm.proValue := FALSE;
    END_IF;
	(* Following bloc checks feedbacksignal of motor *)                           
    fbCheckMotorIsOn((* Inputs *)
                    xSafetyIn           :=  xMotorIsOn,
                    xReferenceIn        :=  xOn OR (xRelease AND xErrorIsOn),
                    (* Parameter *)
                    fbxEnSafetyInput    :=  scParameter.scIO_IsOn.fbxDoesAlarm,
                    fbtStartTime        :=  scParameter.scIO_IsOn.fbtDelayStart,
                    fbtRunTime          :=  scParameter.scIO_IsOn.fbtDelayRun,
                    (* Outputs *)
                    xError              =>  xErrorIsOn);  
                    
    (* Check Motor no error *)
    IF scParameter.scIO_IsNoError.fbxDoesAlarm.proValue > scParameter.scIO_IsNoError.fbxEnable.proValue THEN
        // Alarm Only if Enabled
        scParameter.scIO_IsNoError.fbxDoesAlarm.proValue := FALSE;
    END_IF; 
	(* Following bloc checks errorfeedback of motor *)           
    fbCheckIsError( (* Inputs *)
                    xSafetyIn           :=  xMotorNoError,
                    xReferenceIn        :=  TRUE,
                    (* Parameter *)
                    fbxEnSafetyInput    :=  scParameter.scIO_IsNoError.fbxDoesAlarm,
                    fbtStartTime        :=  scParameter.scIO_IsNoError.fbtDelayStartSps,
                    fbtRunTime          :=  scParameter.scIO_IsNoError.fbtDelayRun,
                    (* Outputs *)
                    xError              =>  xErrorMotorError);     

    xSafetyStopMotor :=  (NOT fbMotor.xHand AND (xErrorMotorError OR xErrorIsOn)) OR xSafetyStop;        
    
    (*Following code scales the controll value to release between the set output parameters*)
    rReleaseScaled  :=  CtaAppBasic.fcScale(    rIn                 :=  rReleaseControllPrio,
                                                rMin                :=  0,
                                                rMax                :=  100,
                                                rOutMin             :=  scParameter.scBase.fbrYMin.proValue,
                                                rOutMax             :=  scParameter.scBase.fbrYMax.proValue);
                                                        
    rReleaseScaled  := LIMIT(scParameter.scBase.fbrYMin.proValue , rReleaseScaled ,scParameter.scBase.fbrYMax.proValue);      
                                  
   (* Lead & run after Time *)
    actVorlaufNachlauf();
    
    (*Following bloc releases the motor and regulates controll value *)                
    fbMotor     (   (* Inputs *)
                    xEn                 :=  xMotorRevisionSwitchOn,
                    xFreigabe           :=  xReleaseMotor,
                    rFreigabeY          :=  rReleaseScaled,
                    xSafetyStop         :=  xSafetyStopMotor,
                    (* Parameter *)
                    fbxEnHandEin        :=  scParameter.scManual.fbxAlowManualOn,
                    fbxGeregelt         :=  scParameter.scBase.fbxRegulatet,
                    fbuiHandMode        :=  scParameter.scManual.fbuiManualState,
                    fbrStellwertHandY   :=  scParameter.scManual.fbrManualOnY,
                    (* Outputs *)
                    xOn                 =>  xOn,
                    rOnY                =>  ,
                    xHand               =>  );
					
	(*Damping of the controll value*)
	fbDumperRonY(	xen		:=	xOn,
					rSoll 	:=	fbMotor.rOnY,
					rY 		=>	rOnY);                
        
    (*Following bloc saves the sarts and operatinghours of the motor*)                                                    
    fbDataCount(	xOperating			    := xOn,
                 	fbudiOperatingStarts	:= scParameter.scData.fbudiOperationStarts,
                 	fbudiOperatingHours		:= scParameter.scData.fbudiOperatingHours);   
                 
    (* EWI *)
    actReport();                 
ELSE
    (* Off if Disabled or Config Error *)
    xOn  := FALSE;
    rOnY := 0;    
    (* Reset Flags *)
    actResetOnDisable();
    IF xConfigError THEN
        (* EWI *)
        actReport();         
	END_IF;
END_IF;

(* State *)
actState();

(* Modbus State *)
actMbState();

(* InfluxDB *)
actTrendLog();

PROPERTY proHandOn : BOOL
SET
IF proHandOn THEN
    scParameter.scManual.fbuiManualState.proValue := 2;
END_IF;
END_SET
GET
proHandOn := xIsHandOn;
END_GET
END_PROPERTY

PROPERTY proAuto : BOOL
SET
IF proAuto THEN
    scParameter.scManual.fbuiManualState.proValue := 0;
END_IF;
END_SET
GET
proAuto := xIsAuto;
END_GET
END_PROPERTY

PROPERTY proHandOff : BOOL
SET
IF proHandOff THEN
    scParameter.scManual.fbuiManualState.proValue := 1;
END_IF;
END_SET
GET
proHandOff := xIsHandOff;
END_GET
END_PROPERTY

PROPERTY proHandOnY : REAL
SET
scParameter.scManual.fbrManualOnY.proValue := proHandOnY;
END_SET
GET
proHandOnY := scParameter.scManual.fbrManualOnY.proValue;
END_GET
END_PROPERTY

PROPERTY proHardWareHandModulAktive : BOOL
GET
proHardWareHandModulAktive := xMotorHand;
END_GET
END_PROPERTY

ACTION actConfig:
(* Config Fb *)
fbConfigFile();

(* Base Parameter *)
scParameter.scBase.fbxEnable                			(_usiParaNr :=  1, ItfConfigFb := fbConfigFile);
scParameter.scBase.fbxRegulatet             			(_usiParaNr :=  2, ItfConfigFb := fbConfigFile);
scParameter.scBase.fbxControllMb            			(_usiParaNr :=  3, ItfConfigFb := fbConfigFile);
scParameter.scBase.fbrYMin                  			(_usiParaNr :=  4, ItfConfigFb := fbConfigFile);
scParameter.scBase.fbrYMax                  			(_usiParaNr :=  5, ItfConfigFb := fbConfigFile);
scParameter.scBase.fbtLeadTime              			(_usiParaNr :=  6, ItfConfigFb := fbConfigFile);
scParameter.scBase.fbtRunAfterTime          			(_usiParaNr :=  7, ItfConfigFb := fbConfigFile);
                                            
(* Fuse Parameter *)                        
scParameter.scFuse.fbxEnable                			(_usiParaNr :=  8, ItfConfigFb := fbconfigFile);
scParameter.scFuse.fbxInputMb               			(_usiParaNr :=  9, ItfConfigFb := fbconfigFile);
scParameter.scFuse.fbxDoesAlarm             			(_usiParaNr := 10, ItfConfigFb := fbconfigFile);
                                            
(* Motor Fuse Parameter *)                  
scParameter.scMotorFuse.fbxEnable           			(_usiParaNr := 11, ItfConfigFb := fbconfigFile);
scParameter.scMotorFuse.fbxInputMb          			(_usiParaNr := 12, ItfConfigFb := fbconfigFile);
scParameter.scMotorFuse.fbxDoesAlarm        			(_usiParaNr := 13, ItfConfigFb := fbconfigFile);
                                            
(* Revision Switch Parameter *)             
scParameter.scIO_RevisionSwitch.fbxEnable  			    (_usiParaNr := 14, ItfConfigFb := fbconfigFile);
scParameter.scIO_RevisionSwitch.fbxInputMb 			    (_usiParaNr := 15, ItfConfigFb := fbconfigFile);
                                            
(* Ready Input Parameter *)                 
scParameter.scIO_IsReady.fbxEnable          		    (_usiParaNr := 16, ItfConfigFb := fbconfigFile);
scParameter.scIO_IsReady.fbxInputMb          			(_usiParaNr := 17, ItfConfigFb := fbconfigFile);
                                            
(* Is On Input Parameter *)                 
scParameter.scIO_IsOn.fbxEnable              			(_usiParaNr := 18, ItfConfigFb := fbconfigFile);
scParameter.scIO_IsOn.fbxInputMb             			(_usiParaNr := 19, ItfConfigFb := fbconfigFile);
scParameter.scIO_IsOn.fbxDoesAlarm           			(_usiParaNr := 20, ItfConfigFb := fbconfigFile);
scParameter.scIO_IsOn.fbtDelayStart          			(_usiParaNr := 21, ItfConfigFb := fbconfigFile);
scParameter.scIO_IsOn.fbtDelayRun            			(_usiParaNr := 22, ItfConfigFb := fbconfigFile);
scParameter.scIO_IsOn.fbiTypeOfAck						(_usiParaNr := 23, ItfConfigFb := fbConfigFile,_MinInit := 1,_MaxInit :=2);
scParameter.scIO_IsOn.fbiMaxErrorRetryAllowed			(_usiParaNr := 24, ItfConfigFb := fbConfigFile); 

(* No Error Input Parameter *)
scParameter.scIO_IsNoError.fbxEnable         			(_usiParaNr := 25, ItfConfigFb := fbconfigFile);
scParameter.scIO_IsNoError.fbxInputMb        			(_usiParaNr := 26, ItfConfigFb := fbconfigFile);
scParameter.scIO_IsNoError.fbxDoesAlarm      			(_usiParaNr := 27, ItfConfigFb := fbconfigFile);
scParameter.scIO_IsNoError.fbtDelayStartSps  			(_usiParaNr := 28, ItfConfigFb := fbconfigFile);
scParameter.scIO_IsNoError.fbtDelayRun       			(_usiParaNr := 29, ItfConfigFb := fbconfigFile);
scParameter.scIO_IsNoError.fbiTypeOfAck					(_usiParaNr := 30, itfConfigFb := fbConfigFile,_MinInit := 1,_MaxInit :=2);
scParameter.scIO_IsNoError.fbiMaxErrorRetryAllowed		(_usiParaNr := 31, itfConfigFb := fbConfigFile);

(* Actual value Input Parameter *)
scParameter.scIO_IsValue.fbxEnable     			        (_usiParaNr := 32, ItfConfigFb := fbconfigFile);
scParameter.scIO_IsValue.fbxInputMb    			        (_usiParaNr := 33, ItfConfigFb := fbconfigFile);
scParameter.scIO_IsValue.fbxDoesAlarm  			        (_usiParaNr := 34, ItfConfigFb := fbconfigFile);
scParameter.scIO_IsValue.fbrMaxDiff    			        (_usiParaNr := 35, ItfConfigFb := fbconfigFile);
scParameter.scIO_IsValue.fbtDelayStart 			        (_usiParaNr := 36, ItfConfigFb := fbconfigFile);
scParameter.scIO_IsValue.fbtDelayRun   			        (_usiParaNr := 37, ItfConfigFb := fbconfigFile);
scParameter.scIO_IsValue.fbiTypeOfAck				    (_usiParaNr := 38, itfConfigFb := fbConfigFile,_MinInit := 0,_MaxInit :=2);
scParameter.scIO_IsValue.fbiMaxErrorRetryAllowed 	    (_usiParaNr := 39, itfConfigFb := fbConfigFile);

(* Manual Parameter *)
scParameter.scManual.fbxAlowManualOn        			(_usiParaNr := 40, ItfConfigFb := fbconfigFile); 
scParameter.scManual.fbuiManualState        			(_usiParaNr := 41, ItfConfigFb := fbconfigFile);
scParameter.scManual.fbrManualOnY           			(_usiParaNr := 42, ItfConfigFb := fbconfigFile);

(* Data Counter *)
scParameter.scData.fbudiOperationStarts     			(_usiParaNr := 43, ItfConfigFb := fbconfigFile);
scParameter.scData.fbudiOperatingHours      			(_usiParaNr := 44, ItfConfigFb := fbconfigFile);

(* Motor Input Hand *)
scParameter.scIO_IsHand.fbxEnable            			(_usiParaNr := 45, ItfConfigFb := fbconfigFile);
scParameter.scIO_IsHand.fbxInputMb           			(_usiParaNr := 46, ItfConfigFb := fbconfigFile);

(* InfluxDb *)
scParameter.scInfluxDb.fbxEnable            			(_usiParaNr := 47, ItfConfigFb := fbconfigFile);

xConfigError := fbConfigFile.xError;
END_ACTION

PROPERTY proConfigError : BOOL
GET
proConfigError := xConfigError;
END_GET
END_PROPERTY

PROPERTY proIconNr : UINT
SET
uiIconNr := proIconNr;
END_SET
GET
proIconNr:= uiIconNr;
END_GET
END_PROPERTY

PROPERTY P_scBase_fbrYMax : CtaSysConfig.ITF_DATATYPE
GET
P_scBase_fbrYMax := scParameter.scBase.fbrYMax;
END_GET
END_PROPERTY

PROPERTY P_scBase_fbrYMin : CtaSysConfig.ITF_DATATYPE
GET
P_scBase_fbrYMin := scParameter.scBase.fbrYMin;
END_GET
END_PROPERTY

PROPERTY P_scBase_fbtLeadTime : CtaSysConfig.ITF_DATATYPE
GET
P_scBase_fbtLeadTime := scParameter.scBase.fbtLeadTime;
END_GET
END_PROPERTY

PROPERTY P_scBase_fbtRunAfterTime : CtaSysConfig.ITF_DATATYPE
GET
P_scBase_fbtRunAfterTime := scParameter.scBase.fbtRunAfterTime;
END_GET
END_PROPERTY

PROPERTY P_scBase_fbxControllMb : CtaSysConfig.ITF_DATATYPE
GET
P_scBase_fbxControllMb := scParameter.scBase.fbxControllMb;
END_GET
END_PROPERTY

PROPERTY P_scBase_fbxEnable : CtaSysConfig.ITF_DATATYPE
GET
P_scBase_fbxEnable := scParameter.scBase.fbxEnable;
END_GET
END_PROPERTY

PROPERTY P_scBase_fbxRegulatet : CtaSysConfig.ITF_DATATYPE
GET
P_scBase_fbxRegulatet := scParameter.scBase.fbxRegulatet;
END_GET
END_PROPERTY

PROPERTY P_scData_fbudiOperatingHours : CtaSysConfig.ITF_DATATYPE
GET
P_scData_fbudiOperatingHours := scParameter.scData.fbudiOperatingHours;
END_GET
END_PROPERTY

PROPERTY P_scData_fbudiOperationStarts : CtaSysConfig.ITF_DATATYPE
GET
P_scData_fbudiOperationStarts := scParameter.scData.fbudiOperationStarts;
END_GET
END_PROPERTY

PROPERTY P_scFuse_fbxDoesAlarm : CtaSysConfig.ITF_DATATYPE
GET
P_scFuse_fbxDoesAlarm := scParameter.scFuse.fbxDoesAlarm;
END_GET
END_PROPERTY

PROPERTY P_scFuse_fbxEnable : CtaSysConfig.ITF_DATATYPE
GET
P_scFuse_fbxEnable := scParameter.scFuse.fbxEnable;
END_GET
END_PROPERTY

PROPERTY P_scFuse_fbxInputMb : CtaSysConfig.ITF_DATATYPE
GET
P_scFuse_fbxInputMb := scParameter.scFuse.fbxInputMb;
END_GET
END_PROPERTY

PROPERTY P_scInfluxDb_fbxEnable : CtaSysConfig.ITF_DATATYPE
GET
P_scInfluxDb_fbxEnable := scParameter.scInfluxDb.fbxEnable;
END_GET
END_PROPERTY

PROPERTY P_scIO_IsHand_fbxEnable : CtaSysConfig.ITF_DATATYPE
GET
P_scIO_IsHand_fbxEnable := scParameter.scIO_IsHand.fbxEnable;
END_GET
END_PROPERTY

PROPERTY P_scIO_IsHand_fbxInputMb : CtaSysConfig.ITF_DATATYPE
GET
P_scIO_IsHand_fbxInputMb := scParameter.scIO_IsHand.fbxInputMb;
END_GET
END_PROPERTY

PROPERTY P_scIO_IsNoError_fbiMaxErrorRetryAllowed : CtaSysConfig.ITF_DATATYPE
GET
P_scIO_IsNoError_fbiMaxErrorRetryAllowed := scParameter.scIO_IsNoError.fbiMaxErrorRetryAllowed;
END_GET
END_PROPERTY

PROPERTY P_scIO_IsNoError_fbiTypeOfAck : CtaSysConfig.ITF_DATATYPE
GET
P_scIO_IsNoError_fbiTypeOfAck := scParameter.scIO_IsNoError.fbiTypeOfAck;
END_GET
END_PROPERTY

PROPERTY P_scIO_IsNoError_fbtDelayRun : CtaSysConfig.ITF_DATATYPE
GET
P_scIO_IsNoError_fbtDelayRun := scParameter.scIO_IsNoError.fbtDelayRun;
END_GET
END_PROPERTY

PROPERTY P_scIO_IsNoError_fbtDelayStartSps : CtaSysConfig.ITF_DATATYPE
GET
P_scIO_IsNoError_fbtDelayStartSps := scParameter.scIO_IsNoError.fbtDelayStartSps;
END_GET
END_PROPERTY

PROPERTY P_scIO_IsNoError_fbxDoesAlarm : CtaSysConfig.ITF_DATATYPE
GET
P_scIO_IsNoError_fbxDoesAlarm := scParameter.scIO_IsNoError.fbxDoesAlarm;
END_GET
END_PROPERTY

PROPERTY P_scIO_IsNoError_fbxEnable : CtaSysConfig.ITF_DATATYPE
GET
P_scIO_IsNoError_fbxEnable := scParameter.scIO_IsNoError.fbxEnable;
END_GET
END_PROPERTY

PROPERTY P_scIO_IsNoError_fbxInputMb : CtaSysConfig.ITF_DATATYPE
GET
P_scIO_IsNoError_fbxInputMb := scParameter.scIO_IsNoError.fbxInputMb;
END_GET
END_PROPERTY

PROPERTY P_scIO_IsOn_fbiMaxErrorRetryAllowed : CtaSysConfig.ITF_DATATYPE
GET
P_scIO_IsOn_fbiMaxErrorRetryAllowed := scParameter.scIO_IsOn.fbiMaxErrorRetryAllowed;
END_GET
END_PROPERTY

PROPERTY P_scIO_IsOn_fbiTypeOfAck : CtaSysConfig.ITF_DATATYPE
GET
P_scIO_IsOn_fbiTypeOfAck := scParameter.scIO_IsOn.fbiTypeOfAck;
END_GET
END_PROPERTY

PROPERTY P_scIO_IsOn_fbtDelayRun : CtaSysConfig.ITF_DATATYPE
GET
P_scIO_IsOn_fbtDelayRun := scParameter.scIO_IsOn.fbtDelayRun;
END_GET
END_PROPERTY

PROPERTY P_scIO_IsOn_fbtDelayStart : CtaSysConfig.ITF_DATATYPE
GET
P_scIO_IsOn_fbtDelayStart := scParameter.scIO_IsOn.fbtDelayStart;
END_GET
END_PROPERTY

PROPERTY P_scIO_IsOn_fbxDoesAlarm : CtaSysConfig.ITF_DATATYPE
GET
P_scIO_IsOn_fbxDoesAlarm := scParameter.scIO_IsOn.fbxDoesAlarm;
END_GET
END_PROPERTY

PROPERTY P_scIO_IsOn_fbxEnable : CtaSysConfig.ITF_DATATYPE
GET
P_scIO_IsOn_fbxEnable := scParameter.scIO_IsOn.fbxEnable;
END_GET
END_PROPERTY

PROPERTY P_scIO_IsOn_fbxInputMb : CtaSysConfig.ITF_DATATYPE
GET
P_scIO_IsOn_fbxInputMb := scParameter.scIO_IsOn.fbxInputMb;
END_GET
END_PROPERTY

PROPERTY P_scIO_IsReady_fbxEnable : CtaSysConfig.ITF_DATATYPE
GET
P_scIO_IsReady_fbxEnable := scParameter.scIO_IsReady.fbxEnable;
END_GET
END_PROPERTY

PROPERTY P_scIO_IsReady_fbxInputMb : CtaSysConfig.ITF_DATATYPE
GET
P_scIO_IsReady_fbxInputMb := scParameter.scIO_IsReady.fbxInputMb;
END_GET
END_PROPERTY

PROPERTY P_scIO_IsValue_fbiMaxErrorRetryAllowed : CtaSysConfig.ITF_DATATYPE
GET
P_scIO_IsValue_fbiMaxErrorRetryAllowed := scParameter.scIO_IsValue.fbiMaxErrorRetryAllowed;
END_GET
END_PROPERTY

PROPERTY P_scIO_IsValue_fbiTypeOfAck : CtaSysConfig.ITF_DATATYPE
GET
P_scIO_IsValue_fbiTypeOfAck := scParameter.scIO_IsValue.fbiTypeOfAck;
END_GET
END_PROPERTY

PROPERTY P_scIO_IsValue_fbrMaxDiff : CtaSysConfig.ITF_DATATYPE
GET
P_scIO_IsValue_fbrMaxDiff := scParameter.scIO_IsValue.fbrMaxDiff;
END_GET
END_PROPERTY

PROPERTY P_scIO_IsValue_fbtDelayRun : CtaSysConfig.ITF_DATATYPE
GET
P_scIO_IsValue_fbtDelayRun := scParameter.scIO_IsValue.fbtDelayRun;
END_GET
END_PROPERTY

PROPERTY P_scIO_IsValue_fbtDelayStart : CtaSysConfig.ITF_DATATYPE
GET
P_scIO_IsValue_fbtDelayStart := scParameter.scIO_IsValue.fbtDelayStart;
END_GET
END_PROPERTY

PROPERTY P_scIO_IsValue_fbxDoesAlarm : CtaSysConfig.ITF_DATATYPE
GET
P_scIO_IsValue_fbxDoesAlarm := scParameter.scIO_IsValue.fbxDoesAlarm;
END_GET
END_PROPERTY

PROPERTY P_scIO_IsValue_fbxEnable : CtaSysConfig.ITF_DATATYPE
GET
P_scIO_IsValue_fbxEnable:= scParameter.scIO_IsValue.fbxEnable;
END_GET
END_PROPERTY

PROPERTY P_scIO_IsValue_fbxInputMb : CtaSysConfig.ITF_DATATYPE
GET
P_scIO_IsValue_fbxInputMb := scParameter.scIO_IsValue.fbxInputMb;
END_GET
END_PROPERTY

PROPERTY P_scIO_RevisionSwitch_fbxEnable : CtaSysConfig.ITF_DATATYPE
GET
P_scIO_RevisionSwitch_fbxEnable := scParameter.scIO_RevisionSwitch.fbxEnable;
END_GET
END_PROPERTY

PROPERTY P_scIO_RevisionSwitch_fbxInputMb : CtaSysConfig.ITF_DATATYPE
GET
P_scIO_RevisionSwitch_fbxInputMb := scParameter.scIO_RevisionSwitch.fbxInputMb;
END_GET
END_PROPERTY

PROPERTY P_scManual_fbrManualOnY : CtaSysConfig.ITF_DATATYPE
GET
P_scManual_fbrManualOnY := scParameter.scManual.fbrManualOnY;
END_GET
END_PROPERTY

PROPERTY P_scManual_fbuiManualState : CtaSysConfig.ITF_DATATYPE
GET
P_scManual_fbuiManualState := scParameter.scManual.fbuiManualState;
END_GET
END_PROPERTY

PROPERTY P_scManual_fbxAlowManualOn : CtaSysConfig.ITF_DATATYPE
GET
P_scManual_fbxAlowManualOn:= scParameter.scManual.fbxAlowManualOn;
END_GET
END_PROPERTY

PROPERTY P_scMotorFuse_fbxDoesAlarm : CtaSysConfig.ITF_DATATYPE
GET
P_scMotorFuse_fbxDoesAlarm := scParameter.scMotorFuse.fbxDoesAlarm;
END_GET
END_PROPERTY

PROPERTY P_scMotorFuse_fbxEnable : CtaSysConfig.ITF_DATATYPE
GET
P_scMotorFuse_fbxEnable := scParameter.scMotorFuse.fbxEnable;
END_GET
END_PROPERTY

PROPERTY P_scMotorFuse_fbxInputMb : CtaSysConfig.ITF_DATATYPE
GET
P_scMotorFuse_fbxInputMb := scParameter.scMotorFuse.fbxInputMb;
END_GET
END_PROPERTY

PROPERTY proRefToRonYDumper : REFERENCE TO CtaAppDumper.fbDumper
GET
proRefToRonYDumper REF= fbDumperRonY;
END_GET
END_PROPERTY

ACTION actMbControll:
IF NOT xModbusTest THEN
    (* Controll Word 0 Digital Controll *)
    (* Release from Modbus *)
    IF scParameter.scBase.fbxControllMb.proValue THEN
        xReleaseFromModBus              := ayMbControllWord[0].0; 
        (* Controll Word 1 setpoint*)
        rReleaseFromModBus              := LIMIT(0,TO_REAL(TO_INT(ayMbControllWord[1]))/10,100);   
    ELSE
        xReleaseFromModBus              := FALSE;
        rReleaseFromModBus              := 0; 
    END_IF;
    (* Motor Ready *)
    IF scParameter.scIO_IsReady.fbxInputMb.proValue THEN
        xInMotorIsReadyMb               := ayMbControllWord[0].2;
    ELSE
        xInMotorIsReadyMb               := FALSE;
    END_IF;
    (* Motor is ON *)
    IF scParameter.scIO_IsOn.fbxInputMb.proValue THEN
        xInMotorIsOnMb                  := ayMbControllWord[0].3;
    ELSE
        xInMotorIsOnMb                  := FALSE;
    END_IF;
    (* Motor no error *)
    IF scParameter.scIO_IsNoError.fbxInputMb.proValue THEN
        xInMotorNoErrorMb               := ayMbControllWord[0].4;
    ELSE
        xInMotorNoErrorMb               := FALSE;
    END_IF;
    (* Revision Switch *)
    IF scParameter.scIO_RevisionSwitch.fbxInputMb.proValue THEN
        xInMotorRevisionSwitchOnMb      := ayMbControllWord[0].5;
    ELSE
        xInMotorRevisionSwitchOnMb      := FALSE;    
    END_IF;
    (* Fuse Ok *)
    IF scParameter.scFuse.fbxInputMb.proValue THEN    
        xInFuseOkMb                     := ayMbControllWord[0].6;
    ELSE
        xInFuseOkMb                     := FALSE;
    END_IF;
    (* Motor Protection *)
    IF scParameter.scMotorFuse.fbxInputMb.proValue THEN
        xInMotorFuseOkMb                := ayMbControllWord[0].7;
    ELSE
        xInMotorFuseOkMb                := FALSE;
    END_IF;
    (* Motor Hand *)
    IF scParameter.scIO_IsHand.fbxInputMb.proValue THEN
        xInMotorHandMb                  := ayMbControllWord[0].8;
    ELSE
        xInMotorHandMb                  := FALSE;
    END_IF;    
ELSE
    xReleaseFromModBus              := FALSE;
    rReleaseFromModBus              := 0;     
    xInMotorIsReadyMb               := FALSE;
    xInMotorIsOnMb                  := FALSE;
    xInMotorNoErrorMb               := FALSE;
    xInMotorRevisionSwitchOnMb      := FALSE; 
    xInFuseOkMb                     := FALSE;
    xInMotorFuseOkMb                := FALSE;
    xInMotorHandMb                  := FALSE;
END_IF;
END_ACTION

ACTION actMbState:
IF NOT xModbusTest THEN
    (* State Word 0 Digital Info*)
    ayMbStateWord[0].00     := xOn;
    ayMbStateWord[0].01     := xIsOn;
    ayMbStateWord[0].02     := xMotorIsReady;
    ayMbStateWord[0].03     := xMotorIsOn;
    ayMbStateWord[0].04     := xMotorNoError;
    ayMbStateWord[0].05     := xMotorRevisionSwitchOn;
    ayMbStateWord[0].06     := xFuseOk;
    ayMbStateWord[0].07     := xMotorFuseOk;
    ayMbStateWord[0].08     := xIsHand;
    ayMbStateWord[0].09     := xIsAuto;
    ayMbStateWord[0].10     := FALSE;
    ayMbStateWord[0].11     := FALSE;
    ayMbStateWord[0].12     := FALSE;
    ayMbStateWord[0].13     := FALSE;
    ayMbStateWord[0].14     := xIsWarning;
    ayMbStateWord[0].15     := xIsError;
    (* State Word 1 setpoint*)
    ayMbStateWord[1]        := TO_WORD((TO_INT(rOnY * 10)));
    (* State Word 2 actual value*)
    ayMbStateWord[2]        := SEL(scParameter.scIO_IsValue.fbxEnable.proValue,TO_WORD((TO_INT(rOnY * 10))),TO_WORD((TO_INT(rInActualValue * 10))));
END_IF;
END_ACTION

PROPERTY proModbusTest : BOOL
SET
xModbusTest := proModbusTest;
END_SET
GET
proModbusTest := xModbusTest;
END_GET
END_PROPERTY

{warning disable C0410}
PROPERTY proModbusStateWord : REFERENCE TO ARRAY[0..3] OF WORD
{warning restore C0410}
GET
proModbusStateWord REF= ayMbStateWord;
END_GET
END_PROPERTY

{warning disable C0410}
PROPERTY proModbusControllWord : REFERENCE TO ARRAY[0..3] OF WORD
{warning restore C0410}
GET
proModbusControllWord REF= ayMbControllWord;
END_GET
END_PROPERTY

PROPERTY proIsOn : BOOL
GET
proIsOn := xIsOn;
END_GET
END_PROPERTY

PROPERTY proIsError : BOOL
GET
proIsError := xIsError;
END_GET
END_PROPERTY

PROPERTY proIsWarning : BOOL
GET
proIsWarning := xIsWarning;
END_GET
END_PROPERTY

PROPERTY proIsRegulatet : BOOL
GET
proIsRegulatet := xIsRegulatet;
END_GET
END_PROPERTY

PROPERTY proIsEnabled : BOOL
GET
proIsEnabled := xIsEnabled;
END_GET
END_PROPERTY

ACTION actState:
xIsWarning        := _xIsWarning;         
xIsError          := _xIsError;          
xIsRegulatet      := scParameter.scBase.fbxRegulatet.proValue;         
xIsEnabled        := scParameter.scBase.fbxEnable.proValue;         
xIsHandOn         := scParameter.scManual.fbuiManualState.proValue = 2;         
xIsHandOff        := scParameter.scManual.fbuiManualState.proValue = 1;          
xIsAuto           := scParameter.scManual.fbuiManualState.proValue = 0 AND NOT xMotorHand;  
xIsHand           := xIsHandOn OR xIsHandOff OR xMotorHand OR xMotorRevisionSwitchOff;
END_ACTION

PROPERTY proMotorIsOn : BOOL
GET
IF scParameter.scIO_IsOn.fbxEnable.proValue THEN
    proMotorIsOn := xMotorIsOn;
ELSE
    proMotorIsOn := xIsOn;
END_IF;
END_GET
END_PROPERTY

PROPERTY proIsHandOnOrOff : BOOL
GET
proIsHandOnOrOff := xIsHand;
END_GET
END_PROPERTY

PROPERTY proIsReady : BOOL
GET
proIsReady := xIsEnabled AND xMotorRevisionSwitchOn AND xMotorIsReady AND NOT xIsError AND NOT xIsHandOff;
END_GET
END_PROPERTY

PROPERTY proLeadTime : TIME
GET
proLeadTime := tLeadTime;
END_GET
END_PROPERTY

PROPERTY proRunAfterTime : TIME
GET
proRunAfterTime := tRunAfter;
END_GET
END_PROPERTY

PROPERTY proIsOnY : REAL
GET
proIsOnY := SEL(scParameter.scIO_IsValue.fbxEnable.proValue,rOnY,rInActualValue);
END_GET
END_PROPERTY

PROPERTY proLeadTimeAktive : BOOL
GET
proLeadTimeAktive := xLeadTimeAktive;
END_GET
END_PROPERTY

PROPERTY proRunAfterTimeAktive : BOOL
GET
proRunAfterTimeAktive := xRunAfterAktive;
END_GET
END_PROPERTY

PROPERTY proRevisionSwitchOk : BOOL
GET
proRevisionSwitchOk := xMotorRevisionSwitchOn;
END_GET
END_PROPERTY

PROPERTY proCountedHours : UDINT
GET
proCountedHours := scParameter.scData.fbudiOperatingHours.proValue;
END_GET
END_PROPERTY

PROPERTY proCountedStarts : UDINT
GET
proCountedStarts := scParameter.scData.fbudiOperationStarts.proValue;
END_GET
END_PROPERTY

PROPERTY proStateSymbol : STRING
GET
IF xIsError THEN
    proStateSymbol := 'CtaVisSymbols.ImagePool.CtaError';
ELSE    
    IF xIsWarning THEN
        IF scEWI.iWarning = 3 THEN
            proStateSymbol := 'CtaVisSymbols.ImagePool.front_hand_Yellow_Off';
        ELSIF scEWI.iWarning = 4 THEN
            proStateSymbol := 'CtaVisSymbols.ImagePool.front_hand_Yellow';
        ELSE
            proStateSymbol := 'CtaVisSymbols.ImagePool.CtaWarning';
        END_IF;
     ELSE
         proStateSymbol := '';
	 END_IF
END_IF;
END_GET
END_PROPERTY

PROPERTY proCountedError : INT
GET
proCountedError := fbReportManager.proAnzError;
END_GET
END_PROPERTY

PROPERTY proCountedInfo : INT
GET
proCountedInfo := fbReportManager.proAnzInfo;
END_GET
END_PROPERTY

PROPERTY proCountedWarning : INT
GET
proCountedWarning := fbReportManager.proAnzWarning;
END_GET
END_PROPERTY

PROPERTY proITF_REPORTMANAGER : CtaAppReport.ITF_REPORTMANAGER
GET
proITF_REPORTMANAGER := fbReportManager;
END_GET
END_PROPERTY

PROPERTY proGetDI_IsOn : BOOL
GET
proGetDI_IsOn := xInMotorIsOn;
END_GET
END_PROPERTY

METHOD metDI_IsOn
VAR_INPUT
	ITF_IN		:	CtaSysIO.ITF_IO;	    
END_VAR
VAR	
	ITF_DI		:	CtaSysIO.ITF_DI;
END_VAR
IF ITF_IN <> 0 THEN
	ITF_MotorIsOn := ITF_IN;	
	IF __QUERYINTERFACE(ITF_MotorIsOn,ITF_DI) THEN		
		xInMotorIsOn := ITF_DI.proValue;
	END_IF	
ELSE
	xInMotorIsOn := FALSE;
END_IF
END_METHOD

PROPERTY proNotShowDI_IsOn : BOOL
GET
proNotShowDI_IsOn := NOT scParameter.scIO_IsOn.fbxEnable.xValue OR scParameter.scIO_IsOn.fbxInputMb.xValue;
END_GET
END_PROPERTY

PROPERTY proIsOn_ITF : CtaSysIO.ITF_IO
GET
proIsOn_ITF := ITF_MotorIsOn;
END_GET
END_PROPERTY

METHOD metDI_RevisionSwitchOk
VAR_INPUT
    ITF_IN		:	CtaSysIO.ITF_IO;
END_VAR
VAR	
	ITF_DI		:	CtaSysIO.ITF_DI;
END_VAR
IF ITF_IN <> 0 THEN	
	ITF_RevisionSwitch := ITF_IN;
	IF __QUERYINTERFACE(ITF_RevisionSwitch,ITF_DI) THEN		
		xInMotorRevisionSwitchOn := ITF_DI.proValue;
	END_IF	
ELSE
	xInMotorRevisionSwitchOn := FALSE;
END_IF
END_METHOD

PROPERTY proNotShowDI_RevisionSwitchOk : BOOL
GET
proNotShowDI_RevisionSwitchOk := NOT scParameter.scIO_RevisionSwitch.fbxEnable.xValue OR scParameter.scIO_RevisionSwitch.fbxInputMb.xValue;
END_GET
END_PROPERTY

PROPERTY proGetDI_RevisionSwitchOK : BOOL
GET
proGetDI_RevisionSwitchOK := xInMotorRevisionSwitchOn;
END_GET
END_PROPERTY

PROPERTY proRevisionSwitch_ITF : CtaSysIO.ITF_IO
GET
proRevisionSwitch_ITF := ITF_RevisionSwitch;
END_GET
END_PROPERTY

METHOD metDI_NoError
VAR_INPUT
    ITF_IN		:	CtaSysIO.ITF_IO;
END_VAR
VAR	
	ITF_DI		:	CtaSysIO.ITF_DI;
END_VAR
IF ITF_IN <> 0 THEN
	ITF_MotorNoError := ITF_IN;	
	IF __QUERYINTERFACE(ITF_MotorNoError,ITF_DI) THEN		
		xInMotorNoError := ITF_DI.proValue;
	END_IF	
ELSE
	xInMotorNoError := FALSE;
END_IF
END_METHOD

PROPERTY proNotShowDI_NoError : BOOL
GET
proNotShowDI_NoError := NOT scParameter.scIO_IsNoError.fbxEnable.xValue OR scParameter.scIO_IsNoError.fbxInputMb.xValue;
END_GET
END_PROPERTY

PROPERTY proGetDI_NoError : BOOL
GET
proGetDI_NoError := xInMotorNoError;
END_GET
END_PROPERTY

PROPERTY proNoError_ITF : CtaSysIO.ITF_IO
GET
proNoError_ITF := ITF_MotorNoError;
END_GET
END_PROPERTY

PROPERTY proGetDI_FuseOK : BOOL
GET
proGetDI_FuseOK := xInFuseOk;
END_GET
END_PROPERTY

METHOD metDI_ITF_FuseOK
VAR_INPUT
	ITF_IN		:	CtaSysIO.ITF_IO;	
END_VAR
VAR
	ITF_DI		:	CtaSysIO.ITF_DI;
END_VAR
IF ITF_IN <> 0 THEN
	ITF_Fuse := ITF_IN; 
	IF __QUERYINTERFACE(ITF_Fuse,ITF_DI) THEN		
		xInFuseOk := ITF_DI.proValue;
	END_IF	
ELSE
	xInFuseOk := FALSE;
END_IF
END_METHOD

PROPERTY proNotShowDI_FuseOk : BOOL
GET
proNotShowDI_FuseOk := NOT scParameter.scFuse.fbxEnable.xValue OR scParameter.scFuse.fbxInputMb.xValue;
END_GET
END_PROPERTY

PROPERTY proFuse_ITF : CtaSysIO.ITF_IO
GET
proFuse_ITF := ITF_Fuse;
END_GET
END_PROPERTY

METHOD metDI_ITF_MotorHand
VAR_INPUT
	ITF_IN		:	CtaSysIO.ITF_IO;	
END_VAR
VAR	
	ITF_DI		:	CtaSysIO.ITF_DI;
END_VAR
IF ITF_IN <> 0 THEN	
	ITF_MotorHand := ITF_IN;
	IF __QUERYINTERFACE(ITF_MotorHand,ITF_DI) THEN		
		xMotorHand := ITF_DI.proValue;
	END_IF	
ELSE
	xMotorHand := FALSE;
END_IF
END_METHOD

PROPERTY proNotShowDI_MotorHand : BOOL
GET
proNotShowDI_MotorHand := NOT scParameter.scIO_IsHand.fbxEnable.xValue OR scParameter.scIO_IsHand.fbxInputMb.xValue;
END_GET
END_PROPERTY

PROPERTY proGetDI_MotorHand : BOOL
GET
proGetDI_MotorHand := xInMotorHand;
END_GET
END_PROPERTY

PROPERTY proHandModul_ITF : CtaSysIO.ITF_IO
GET
proHandModul_ITF := ITF_MotorHand;
END_GET
END_PROPERTY

METHOD metDI_IsReady
VAR_INPUT
    ITF_IN		:	CtaSysIO.ITF_IO;
END_VAR
VAR	
	ITF_DI		:	CtaSysIO.ITF_DI;
END_VAR
IF ITF_IN <> 0 THEN	
	ITF_MotorIsReady := ITF_IN;
	IF __QUERYINTERFACE(ITF_MotorIsReady,ITF_DI) THEN		
		xInMotorIsReady := ITF_DI.proValue;
	END_IF	
ELSE
	xInMotorIsReady := FALSE;
END_IF
END_METHOD

PROPERTY proNotShowDI_Ready : BOOL
GET
proNotShowDI_Ready := NOT scParameter.scIO_IsReady.fbxEnable.xValue OR scParameter.scIO_IsReady.fbxInputMb.xValue;
END_GET
END_PROPERTY

PROPERTY proGetDI_IsReady : BOOL
GET
proGetDI_IsReady := xInMotorIsReady;
END_GET
END_PROPERTY

PROPERTY proReady_ITF : CtaSysIO.ITF_IO
GET
proReady_ITF := ITF_MotorIsReady;
END_GET
END_PROPERTY

METHOD metDI_MotorFuseOk
VAR_INPUT
    ITF_IN		:	CtaSysIO.ITF_IO;
END_VAR
VAR	
	ITF_DI		:	CtaSysIO.ITF_DI;
END_VAR
IF ITF_IN <> 0 THEN
	ITF_MotorFuse := ITF_IN;	
	IF __QUERYINTERFACE(ITF_MotorFuse,ITF_DI) THEN		
		xInMotorFuseOk := ITF_DI.proValue;
	END_IF	
ELSE
	xInMotorFuseOk := FALSE;
END_IF
END_METHOD

PROPERTY proNotShowDI_MotorFuseOk : BOOL
GET
proNotShowDI_MotorFuseOk := NOT scParameter.scMotorFuse.fbxEnable.xValue OR scParameter.scMotorFuse.fbxInputMb.xValue;
END_GET
END_PROPERTY

PROPERTY proGetDI_MotorFuseOk : BOOL
GET
proGetDI_MotorFuseOk := xInMotorFuseOk;
END_GET
END_PROPERTY

PROPERTY proMotorFuse_ITF : CtaSysIO.ITF_IO
GET
proMotorFuse_ITF := ITF_MotorFuse;
END_GET
END_PROPERTY

METHOD metDO_On : BOOL
VAR_INPUT
    ITF_IN		:	CtaSysIO.ITF_IO;
END_VAR
VAR	
	ITF_DO		:	CtaSysIO.ITF_DO;
END_VAR
IF ITF_IN <> 0 THEN	
	ITF_xOn := ITF_IN;
	IF __QUERYINTERFACE(ITF_xOn,ITF_DO) THEN		
		ITF_DO.proValue := xOn;
	END_IF	
ELSE
	metDO_On := xOn;
END_IF
END_METHOD

PROPERTY proOn_ITF : CtaSysIO.ITF_IO
GET
proOn_ITF := ITF_xOn;
END_GET
END_PROPERTY

METHOD metAO_OnY : REAL
VAR_INPUT
    ITF_IN		:	CtaSysIO.ITF_IO;
END_VAR
VAR	
	ITF_AO		:	CtaSysIO.ITF_AO;
END_VAR
IF ITF_IN <> 0 THEN
	ITF_rOnY := ITF_IN;	
	IF __QUERYINTERFACE(ITF_rOnY,ITF_AO) THEN		
		ITF_AO.proValue := rOnY;
	END_IF	
ELSE
	metAO_OnY := rOnY;
END_IF
END_METHOD

PROPERTY proOnY_ITF : CtaSysIO.ITF_IO
GET
proOnY_ITF := ITF_rOnY;
END_GET
END_PROPERTY

PROPERTY proNotShowAI_ActualValue : BOOL
GET
proNotShowAI_ActualValue := NOT scParameter.scIO_IsValue.fbxEnable.xValue OR scParameter.scIO_IsValue.fbxInputMb.xValue;
END_GET
END_PROPERTY

METHOD metAI_ActualValue
VAR_INPUT
    ITF_IN		:	CtaSysIO.ITF_IO;
END_VAR
VAR	
	ITF_AI		:	CtaSysIO.ITF_AI;
END_VAR
IF ITF_IN <> 0 THEN
	ITF_ActualValue := ITF_IN;	
	IF __QUERYINTERFACE(ITF_ActualValue,ITF_AI) THEN		
		rInActualValue := ITF_AI.proValue;
	END_IF	
ELSE
	rInActualValue := 0;
END_IF
END_METHOD

PROPERTY proGetAI_ActualValue : REAL
GET
proGetAI_ActualValue := rInActualValue;
END_GET
END_PROPERTY

PROPERTY proActualValue_ITF : CtaSysIO.ITF_IO
GET
proActualValue_ITF := ITF_ActualValue;
END_GET
END_PROPERTY

PROPERTY proOnY : REAL
GET
proOnY := rOnY;
END_GET
END_PROPERTY

PROPERTY proOn : BOOL
GET
proOn := xOn;
END_GET
END_PROPERTY

ACTION actVorlaufNachlauf:
(* Lead Time *)
TON_LeadTime (  IN  :=  xOn,
                PT  :=  scParameter.scBase.fbtLeadTime.proValue);
            
IF xOn AND TON_LeadTime.ET <> T#0S AND TON_LeadTime.ET <> scParameter.scBase.fbtLeadTime.proValue THEN                
    tLeadTime       := scParameter.scBase.fbtLeadTime.proValue - TON_LeadTime.ET;    
    xLeadTimeAktive := TRUE; 
ELSE
    tLeadTime       := T#0S;
    xLeadTimeAktive := FALSE; 
END_IF;
(* State is On *)    
IF scParameter.scIO_IsOn.fbxEnable.proValue AND scParameter.scIO_IsOn.fbxDoesAlarm.proValue THEN
    xIsOn := fbCheckMotorIsOn.proOK AND (TON_LeadTime.Q OR xRunAfterAktive);
ELSE
    xIsOn := TON_LeadTime.Q OR xRunAfterAktive;
END_IF;         
(* Run After Time *)

TOF_RunAfter(   IN  :=  xReleaseControllPrio,
                PT  :=  scParameter.scBase.fbtRunAfterTime.proValue,
                Q   =>  xReleaseMotor);    
 
IF NOT xRelease AND xOn AND TOF_RunAfter.Q THEN                
    tRunAfter       := scParameter.scBase.fbtRunAfterTime.proValue - TOF_RunAfter.ET;  
	
    xRunAfterAktive := TRUE; 
    TON_LeadTime.PT  := T#0MS;
    TON_LeadTime.IN  := FALSE ;  
    TON_LeadTime();  	
ELSE
    tRunAfter       := T#0S;
    xRunAfterAktive := FALSE; 
END_IF;  
(* Reset on Safety Stopp *)
IF xSafetyStopMotor THEN
    TON_LeadTime.PT  := T#0MS;
    TON_LeadTime.IN  := FALSE ;  
    TON_LeadTime();  
    xLeadTimeAktive := FALSE;
    TOF_RunAfter.PT := T#0MS;
    TOF_RunAfter.IN := FALSE ;  
    TOF_RunAfter();  
    xRunAfterAktive := FALSE;    
    xReleaseMotor   := FALSE;
    xIsOn           := FALSE;
END_IF;
END_ACTION

ACTION actPrioOfControll:
(* get Controll request *)
xReleaseControllPrio := SEL(xRelease,xReleaseFromModBus,xRelease);  // xRelease request from Software has prio
rReleaseControllPrio := SEL(xRelease,rReleaseFromModBus,rRelease);  // rRelease request from Software has prio

(* Get state from Input or ModBus *)
(* Fuse ok *)
// Flag FuseOk True if not Enabled
xFuseOk                            := SEL(scParameter.scFuse.fbxEnable.xValue                   ,TRUE   ,SEL(scParameter.scFuse.fbxInputMb.xValue               ,xInFuseOk                  ,xInFuseOkMb                ));                     
(* Motor fuse ok *)
// Flag MotorFuseOk True if not Enabled
xMotorFuseOk                       := SEL(scParameter.scMotorFuse.fbxEnable.xValue              ,TRUE   ,SEL(scParameter.scMotorFuse.fbxInputMb.xValue          ,xInMotorFuseOk             ,xInMotorFuseOkMb           ));
(* Motor no error *)
// Flag MotorNoError True if not Enabled
xMotorNoError                      := SEL(scParameter.scIO_IsNoError.fbxEnable.xValue            ,TRUE   ,SEL(scParameter.scIO_IsNoError.fbxInputMb.xValue        ,xInMotorNoError            ,xInMotorNoErrorMb          ));
(* Motor is ready *)
// Flag MotorIsReady True if not Enabled
xMotorIsReady                      := SEL(scParameter.scIO_IsReady.fbxEnable.xValue              ,TRUE   ,SEL(scParameter.scIO_IsReady.fbxInputMb.xValue          ,xInMotorIsReady            ,xInMotorIsReadyMb          )); 
(* Revision Switch *)
// Flag MotorRevisionSwitchOn True if not Enabled
xMotorRevisionSwitchOn             := SEL(scParameter.scIO_RevisionSwitch.fbxEnable.xValue     ,TRUE   ,SEL(scParameter.scIO_RevisionSwitch.fbxInputMb.xValue ,xInMotorRevisionSwitchOn   ,xInMotorRevisionSwitchOnMb ));
xMotorRevisionSwitchOff            := NOT xMotorRevisionSwitchOn;
(* Motor is on *)
// Flag MotorIsOn False if not Enabled
xMotorIsOn                         := SEL(scParameter.scIO_IsOn.fbxEnable.xValue                 ,FALSE  ,SEL(scParameter.scIO_IsOn.fbxInputMb.xValue             ,xInMotorIsOn               ,xInMotorIsOnMb             ));  
(* Motor is hand *)
// Flag MotorHand False if not Enabled
xMotorHand                         := SEL(scParameter.scIO_IsHand.fbxEnable.xValue               ,FALSE  ,SEL(scParameter.scIO_IsHand.fbxInputMb.xValue           ,xInMotorHand               ,xInMotorHandMb             ));
END_ACTION

ACTION actResetOnDisable:
(* Reset Lead and Run After Command *)
    TON_LeadTime.PT                 := T#0MS;
    TON_LeadTime.IN                 := FALSE ;  
    TON_LeadTime();  
    xLeadTimeAktive                 := FALSE;
    TOF_RunAfter.PT                 := T#0MS;
    TOF_RunAfter.IN                 := FALSE ;  
    TOF_RunAfter();                  
    xRunAfterAktive                 := FALSE;    
    xReleaseMotor                   := FALSE;
    xIsOn                           := FALSE;
    xFuseOk                         := FALSE;    
    xMotorFuseOk                    := FALSE;
    xMotorNoError                   := FALSE;
    xMotorIsReady                   := FALSE;
    xMotorRevisionSwitchOn          := FALSE;
    xMotorIsOn                      := FALSE;
    xMotorHand                      := FALSE;
END_ACTION

PROPERTY proEn : BOOL
SET
xIsEnabled := proEn;
END_SET
GET
proEn := xIsEnabled;
END_GET
END_PROPERTY

PROPERTY proEnSymbol : STRING
GET
IF xIsEnabled THEN
    proEnSymbol := 'CtaVisSymbols.ImagePool.CheckboxChecked_blue';
ELSE    
    proEnSymbol := 'CtaVisSymbols.ImagePool.CheckboxUnchecked_withe'; 
END_IF;
END_GET
END_PROPERTY

ACTION actTrendLog:
(* Schaltbefehl *)
fbTrendxOn.ENABLE 			:= 	scParameter.scBase.fbxEnable.proValue AND 
								scParameter.scInfluxDb.fbxEnable.proValue;
fbTrendxOn.KEY				:= 	CONCAT(stObjID,'_xOn');
fbTrendxOn.SET_VALUE		:= 	xOn;
	
(* Betriebsmeldung *)
fbTrendxIsOn.ENABLE			:= 	scParameter.scBase.fbxEnable.proValue AND 
								scParameter.scInfluxDb.fbxEnable.proValue;
fbTrendxIsOn.KEY			:= 	CONCAT(stObjID,'_xIsOn');
fbTrendxIsOn.SET_VALUE		:= 	xIsOn;
							  
(* Betriebsmeldung Motor*)
fbTrendxMotorIsOn.ENABLE	:=	scParameter.scBase.fbxEnable.proValue AND 
								scParameter.scInfluxDb.fbxEnable.proValue;
fbTrendxMotorIsOn.KEY		:= 	CONCAT(stObjID,'_xMotorIsOn');
fbTrendxMotorIsOn.SET_VALUE	:= 	xMotorIsOn;

(* Stellwert*)
fbTrendrOnY.ENABLE 			:=	scParameter.scBase.fbxEnable.proValue AND 
								scParameter.scInfluxDb.fbxEnable.proValue;
fbTrendrOnY.KEY				:= 	CONCAT(stObjID,'_rOnY');
fbTrendrOnY.SET_VALUE		:= 	rOnY;		

(* Istwert*)
fbTrendrIsOnY.ENABLE		:= 	scParameter.scBase.fbxEnable.proValue AND 
								scParameter.scInfluxDb.fbxEnable.proValue;
fbTrendrIsOnY.KEY			:= 	CONCAT(stObjID,'_rIsOnY');
fbTrendrIsOnY.SET_VALUE		:= 	proIsOnY;

(* Fehler*)
fbTrendxError.ENABLE		:= 	scParameter.scBase.fbxEnable.proValue AND 
								scParameter.scInfluxDb.fbxEnable.proValue;
fbTrendxError.KEY			:= 	CONCAT(stObjID,'_xError');
fbTrendxError.SET_VALUE		:= 	xIsError;
END_ACTION

ACTION actReport:
(* EWI Manager *)
fbReportManager(	stErrorInitReportTextListIn		:=	ADR(GlobalKonstant.stReportTextListError),
					stWarningInitReportTextListIn	:=	ADR(GlobalKonstant.stReportTextListWarning),
					stInfoInitReportTextListIn		:=	ADR(GlobalKonstant.stReportTextListInfo),
					scReportNr						:=	scEWI);
(* Errors *)                        
        (* Meldung Error On *)
        ayErrorReporter[1].proPrio  := 3;
        ayErrorReporter[1].metReport(     		xSetReportIn					:= xErrorIsOn AND scParameter.scIO_IsOn.fbxDoesAlarm.proValue AND scParameter.scIO_IsOn.fbxEnable.proValue,
												iReportID						:= 1,
												enReportTypeIn					:= CtaAppReport.enReportType.Error,  
												enReportAcknowledgeTypeIn   	:= scParameter.scIO_IsOn.fbiTypeOfAck.proValue,
												tDelay							:= T#0S, 
												ITF_BMK_IN						:= THIS^,			              
												pstReportTextListIn				:= ADR(GlobalKonstant.stReportTextListError),
												stOptionalReportText		    := '',   
												iRetryTilReportLock 		    := scParameter.scIO_IsOn.fbiMaxErrorRetryAllowed.proValue, 
												xResetCount         		    := FALSE,  
												tReset						    := T#24H); 		

        (* Error Motor *)    
        ayErrorReporter[2].proPrio  := 3;
        ayErrorReporter[2].metReport(     		xSetReportIn					:= xErrorMotorError AND scParameter.scIO_IsNoError.fbxDoesAlarm.proValue AND scParameter.scIO_IsNoError.fbxEnable.proValue,
												iReportID						:= 2,
												enReportTypeIn					:= CtaAppReport.enReportType.Error,  
												enReportAcknowledgeTypeIn   	:= scParameter.scIO_IsNoError.fbiTypeOfAck.proValue,
												tDelay							:= T#0S, 
												ITF_BMK_IN						:= THIS^,			              
												pstReportTextListIn				:= ADR(GlobalKonstant.stReportTextListError),
												stOptionalReportText		    := '',   
												iRetryTilReportLock 		    := scParameter.scIO_IsNoError.fbiMaxErrorRetryAllowed.proValue, 
												xResetCount         		    := FALSE,  
												tReset						    := T#24H); 	  
                           
        (* Error Fuse *) 
        ayErrorReporter[3].proPrio  := 2;   
        ayErrorReporter[3].metReport(     		xSetReportIn					:= NOT xFuseOk AND scParameter.scFuse.fbxDoesAlarm.proValue AND scParameter.scFuse.fbxEnable.proValue,
												iReportID						:= 3,
												enReportTypeIn					:= CtaAppReport.enReportType.Error,  
												enReportAcknowledgeTypeIn   	:= CtaAppReport.enReportacknowledgeType.Auto,
												tDelay							:= T#1S, 
												ITF_BMK_IN						:= THIS^,			              
												pstReportTextListIn				:= ADR(GlobalKonstant.stReportTextListError),
												stOptionalReportText		    := '',   
												iRetryTilReportLock 		    := 0, 
												xResetCount         		    := FALSE,  
												tReset						    := T#24H);
                                                
        (* Error Motor Fuse *)    
        ayErrorReporter[4].proPrio  := 2;
        ayErrorReporter[4].metReport(     		xSetReportIn					:= NOT xMotorFuseOk AND scParameter.scMotorFuse.fbxDoesAlarm.proValue AND scParameter.scMotorFuse.fbxEnable.proValue,
												iReportID						:= 4,
												enReportTypeIn					:= CtaAppReport.enReportType.Error,  
												enReportAcknowledgeTypeIn   	:= CtaAppReport.enReportacknowledgeType.Auto,
												tDelay							:= T#1S, 
												ITF_BMK_IN						:= THIS^,			              
												pstReportTextListIn				:= ADR(GlobalKonstant.stReportTextListError),
												stOptionalReportText		    := '',   
												iRetryTilReportLock 		    := 0, 
												xResetCount         		    := FALSE,  
												tReset						    := T#24H);                                                

        (* Config Error *)    
        ayErrorReporter[5].proPrio  := 1;
        ayErrorReporter[5].metReport(     		xSetReportIn					:= xConfigError,
												iReportID						:= 5,
												enReportTypeIn					:= CtaAppReport.enReportType.Error,  
												enReportAcknowledgeTypeIn   	:= CtaAppReport.enReportacknowledgeType.Quit,
												tDelay							:= T#1S, 
												ITF_BMK_IN						:= THIS^,			              
												pstReportTextListIn				:= ADR(GlobalKonstant.stReportTextListError),
												stOptionalReportText		    := '',   
												iRetryTilReportLock 		    := 0, 
												xResetCount         		    := FALSE,  
												tReset						    := T#24H);                                           
(* Warnungen *)      
        (* Warnung Sicherheits Stopp *)      
        ayWarningReporter[1].proPrio := 2;
        ayWarningReporter[1].metReport(			xSetReportIn					:= xSafetyStopMotor AND xReleaseMotor,
												iReportID						:= 1,
												enReportTypeIn					:= CtaAppReport.enReportType.Warning,  
												enReportAcknowledgeTypeIn   	:= CtaAppReport.enReportAcknowledgeType.Auto,
												tDelay							:= T#0S, 
												ITF_BMK_IN						:= THIS^,			              
												pstReportTextListIn				:= ADR(GlobalKonstant.stReportTextListWarning),
												stOptionalReportText		    := '',   
												iRetryTilReportLock 		    := 0, 
												xResetCount         		    := FALSE,  
												tReset						    := T#24H);                       
                                  
        (* Warnung Revisionsschalter Aus *)
        ayWarningReporter[2].proPrio := 1;
	    ayWarningReporter[2].proHandLokal :=    xMotorRevisionSwitchOff; 
        ayWarningReporter[2].metReport(			xSetReportIn					:= xMotorRevisionSwitchOff,
												iReportID						:= 2,
												enReportTypeIn					:= CtaAppReport.enReportType.Warning,  
												enReportAcknowledgeTypeIn   	:= CtaAppReport.enReportAcknowledgeType.Auto,
												tDelay							:= T#0S, 
												ITF_BMK_IN						:= THIS^,			              
												pstReportTextListIn				:= ADR(GlobalKonstant.stReportTextListWarning),
												stOptionalReportText		    := '',   
												iRetryTilReportLock 		    := 0, 
												xResetCount         		    := FALSE,  
												tReset						    := T#24H);     

        (* Warnung Hand Aus *)      
        ayWarningReporter[3].proPrio := 3;  
		ayWarningReporter[3].proHandLokal :=    xIsHandOff; 
        ayWarningReporter[3].metReport(			xSetReportIn					:= xIsHandOff,
												iReportID						:= 3,
												enReportTypeIn					:= CtaAppReport.enReportType.Warning,  
												enReportAcknowledgeTypeIn   	:= CtaAppReport.enReportAcknowledgeType.Auto,
												tDelay							:= T#0S, 
												ITF_BMK_IN						:= THIS^,			              
												pstReportTextListIn				:= ADR(GlobalKonstant.stReportTextListWarning),
												stOptionalReportText		    := '',   
												iRetryTilReportLock 		    := 0, 
												xResetCount         		    := FALSE,  
												tReset						    := T#24H);                                  
                                
        (* Warnung Hand Ein *)    
        ayWarningReporter[4].proPrio := 3; 
		ayWarningReporter[4].proHandLokal :=    xIsHandOn;
        ayWarningReporter[4].metReport(			xSetReportIn					:= xIsHandOn,
												iReportID						:= 4,
												enReportTypeIn					:= CtaAppReport.enReportType.Warning,  
												enReportAcknowledgeTypeIn   	:= CtaAppReport.enReportAcknowledgeType.Auto,
												tDelay							:= T#0S, 
												ITF_BMK_IN						:= THIS^,			              
												pstReportTextListIn				:= ADR(GlobalKonstant.stReportTextListWarning),
												stOptionalReportText		    := '',   
												iRetryTilReportLock 		    := 0, 
												xResetCount         		    := FALSE,  
												tReset						    := T#24H);   
 
        (* Warnung Handmodul Motor *)   
        ayWarningReporter[5].proPrio := 4;  
		ayWarningReporter[5].proHandLokal :=    xMotorHand;
        ayWarningReporter[5].metReport(			xSetReportIn					:= xMotorHand,
												iReportID						:= 5,
												enReportTypeIn					:= CtaAppReport.enReportType.Warning,  
												enReportAcknowledgeTypeIn   	:= CtaAppReport.enReportAcknowledgeType.Auto,
												tDelay							:= T#0S, 
												ITF_BMK_IN						:= THIS^,			              
												pstReportTextListIn				:= ADR(GlobalKonstant.stReportTextListWarning),
												stOptionalReportText		    := '',   
												iRetryTilReportLock 		    := 0, 
												xResetCount         		    := FALSE,  
												tReset						    := T#24H);                                                   
(* Sync Reports *)                                         
FOR difor := LOWER_BOUND(ayErrorReporter,1) TO UPPER_BOUND(ayErrorReporter,1) DO
	fbReportManager.metSyncReporter(ayErrorReporter[difor]);	
END_FOR;
FOR difor := LOWER_BOUND(ayWarningReporter,1) TO UPPER_BOUND(ayWarningReporter,1) DO
	fbReportManager.metSyncReporter(ayWarningReporter[difor]);	
END_FOR;
                                                                             
_xIsError   := scEWI.iError <> 0;
_xIsWarning := scEWI.iWarning <> 0;
END_ACTION

{attribute 'monitoring' := 'variable'}
PROPERTY proLockDown : BOOL
GET
proLockDown := proIsError;
END_GET
END_PROPERTY

{attribute 'monitoring' := 'variable'}
PROPERTY proAvailable : BOOL
GET
proAvailable := proIsReady;
END_GET
END_PROPERTY

{attribute 'monitoring' := 'variable'}
PROPERTY proAcknowlege : BOOL
GET
proAcknowlege := proIsOn;
END_GET
END_PROPERTY

END_FUNCTION_BLOCK

// 21 Interface/ITF_ANTRIEB
INTERFACE ITF_ANTRIEB EXTENDS CtaAppBmk.ITF_BMK , CtaAppModbusSpezifikation.ITF_MODBUS_SPEZIFIKATION

{attribute 'hide'} 
PROPERTY INTERNAL proModbusTest : BOOL
GET
END_GET
SET
END_SET
END_PROPERTY

{warning disable C0410}
PROPERTY proModbusStateWord : REFERENCE TO ARRAY[0..3] OF WORD
{warning restore C0410}
GET
END_GET
END_PROPERTY

{warning disable C0410}
PROPERTY proModbusControllWord : REFERENCE TO ARRAY[0..3] OF WORD
{warning restore C0410}
GET
END_GET
END_PROPERTY

{attribute 'hide'} 
PROPERTY proConfigError : BOOL
GET
END_GET
END_PROPERTY

PROPERTY P_scIO_IsHand_fbxEnable : CtaSysConfig.ITF_DATATYPE
GET
END_GET
END_PROPERTY

PROPERTY P_scIO_IsHand_fbxInputMb : CtaSysConfig.ITF_DATATYPE
GET
END_GET
END_PROPERTY

PROPERTY P_scIO_IsNoError_fbxEnable : CtaSysConfig.ITF_DATATYPE
GET
END_GET
END_PROPERTY

PROPERTY P_scIO_IsNoError_fbxInputMb : CtaSysConfig.ITF_DATATYPE
GET
END_GET
END_PROPERTY

PROPERTY P_scIO_IsNoError_fbxDoesAlarm : CtaSysConfig.ITF_DATATYPE
GET
END_GET
END_PROPERTY

PROPERTY P_scIO_IsNoError_fbtDelayStartSps : CtaSysConfig.ITF_DATATYPE
GET
END_GET
END_PROPERTY

PROPERTY P_scIO_IsNoError_fbtDelayRun : CtaSysConfig.ITF_DATATYPE
GET
END_GET
END_PROPERTY

PROPERTY P_scIO_IsNoError_fbiTypeOfAck : CtaSysConfig.ITF_DATATYPE
GET
END_GET
END_PROPERTY

PROPERTY P_scIO_IsNoError_fbiMaxErrorRetryAllowed : CtaSysConfig.ITF_DATATYPE
GET
END_GET
END_PROPERTY

PROPERTY P_scIO_IsOn_fbxInputMb : CtaSysConfig.ITF_DATATYPE
GET
END_GET
END_PROPERTY

PROPERTY P_scIO_IsOn_fbxEnable : CtaSysConfig.ITF_DATATYPE
GET
END_GET
END_PROPERTY

PROPERTY P_scIO_IsOn_fbtDelayStart : CtaSysConfig.ITF_DATATYPE
GET
END_GET
END_PROPERTY

PROPERTY P_scIO_IsOn_fbxDoesAlarm : CtaSysConfig.ITF_DATATYPE
GET
END_GET
END_PROPERTY

PROPERTY P_scIO_IsOn_fbtDelayRun : CtaSysConfig.ITF_DATATYPE
GET
END_GET
END_PROPERTY

PROPERTY P_scIO_IsOn_fbiTypeOfAck : CtaSysConfig.ITF_DATATYPE
GET
END_GET
END_PROPERTY

PROPERTY P_scIO_IsOn_fbiMaxErrorRetryAllowed : CtaSysConfig.ITF_DATATYPE
GET
END_GET
END_PROPERTY

PROPERTY P_scIO_IsReady_fbxEnable : CtaSysConfig.ITF_DATATYPE
GET
END_GET
END_PROPERTY

PROPERTY P_scIO_IsReady_fbxInputMb : CtaSysConfig.ITF_DATATYPE
GET
END_GET
END_PROPERTY

PROPERTY P_scIO_IsValue_fbxInputMb : CtaSysConfig.ITF_DATATYPE
GET
END_GET
END_PROPERTY

PROPERTY P_scIO_IsValue_fbxEnable : CtaSysConfig.ITF_DATATYPE
GET
END_GET
END_PROPERTY

PROPERTY P_scIO_IsValue_fbxDoesAlarm : CtaSysConfig.ITF_DATATYPE
GET
END_GET
END_PROPERTY

PROPERTY P_scIO_IsValue_fbtDelayStart : CtaSysConfig.ITF_DATATYPE
GET
END_GET
END_PROPERTY

PROPERTY P_scIO_IsValue_fbtDelayRun : CtaSysConfig.ITF_DATATYPE
GET
END_GET
END_PROPERTY

PROPERTY P_scIO_IsValue_fbiTypeOfAck : CtaSysConfig.ITF_DATATYPE
GET
END_GET
END_PROPERTY

PROPERTY P_scIO_IsValue_fbiMaxErrorRetryAllowed : CtaSysConfig.ITF_DATATYPE
GET
END_GET
END_PROPERTY

PROPERTY P_scIO_IsValue_fbrMaxDiff : CtaSysConfig.ITF_DATATYPE
GET
END_GET
END_PROPERTY

PROPERTY P_scIO_RevisionSwitch_fbxEnable : CtaSysConfig.ITF_DATATYPE
GET
END_GET
END_PROPERTY

PROPERTY P_scIO_RevisionSwitch_fbxInputMb : CtaSysConfig.ITF_DATATYPE
GET
END_GET
END_PROPERTY

PROPERTY P_scBase_fbxEnable : CtaSysConfig.ITF_DATATYPE
GET
END_GET
END_PROPERTY

PROPERTY P_scBase_fbxRegulatet : CtaSysConfig.ITF_DATATYPE
GET
END_GET
END_PROPERTY

PROPERTY P_scBase_fbxControllMb : CtaSysConfig.ITF_DATATYPE
GET
END_GET
END_PROPERTY

PROPERTY P_scBase_fbrYMin : CtaSysConfig.ITF_DATATYPE
GET
END_GET
END_PROPERTY

PROPERTY P_scBase_fbrYMax : CtaSysConfig.ITF_DATATYPE
GET
END_GET
END_PROPERTY

PROPERTY P_scBase_fbtLeadTime : CtaSysConfig.ITF_DATATYPE
GET
END_GET
END_PROPERTY

PROPERTY P_scBase_fbtRunAfterTime : CtaSysConfig.ITF_DATATYPE
GET
END_GET
END_PROPERTY

PROPERTY P_scFuse_fbxEnable : CtaSysConfig.ITF_DATATYPE
GET
END_GET
END_PROPERTY

PROPERTY P_scFuse_fbxInputMb : CtaSysConfig.ITF_DATATYPE
GET
END_GET
END_PROPERTY

PROPERTY P_scFuse_fbxDoesAlarm : CtaSysConfig.ITF_DATATYPE
GET
END_GET
END_PROPERTY

PROPERTY P_scMotorFuse_fbxInputMb : CtaSysConfig.ITF_DATATYPE
GET
END_GET
END_PROPERTY

PROPERTY P_scMotorFuse_fbxEnable : CtaSysConfig.ITF_DATATYPE
GET
END_GET
END_PROPERTY

PROPERTY P_scMotorFuse_fbxDoesAlarm : CtaSysConfig.ITF_DATATYPE
GET
END_GET
END_PROPERTY

PROPERTY P_scManual_fbxAlowManualOn : CtaSysConfig.ITF_DATATYPE
GET
END_GET
END_PROPERTY

PROPERTY P_scManual_fbuiManualState : CtaSysConfig.ITF_DATATYPE
GET
END_GET
END_PROPERTY

PROPERTY P_scManual_fbrManualOnY : CtaSysConfig.ITF_DATATYPE
GET
END_GET
END_PROPERTY

PROPERTY P_scInfluxDb_fbxEnable : CtaSysConfig.ITF_DATATYPE
GET
END_GET
END_PROPERTY

PROPERTY P_scData_fbudiOperationStarts : CtaSysConfig.ITF_DATATYPE
GET
END_GET
END_PROPERTY

PROPERTY P_scData_fbudiOperatingHours : CtaSysConfig.ITF_DATATYPE
GET
END_GET
END_PROPERTY

PROPERTY proRefToRonYDumper : REFERENCE TO CtaAppDumper.fbDumper
GET
END_GET
END_PROPERTY

{attribute 'hide'} 
PROPERTY INTERNAL proCountedError : INT
GET
END_GET
END_PROPERTY

{attribute 'hide'} 
PROPERTY INTERNAL proCountedInfo : INT
GET
END_GET
END_PROPERTY

{attribute 'hide'} 
PROPERTY INTERNAL proITF_REPORTMANAGER : CtaAppReport.ITF_REPORTMANAGER
GET
END_GET
END_PROPERTY

{attribute 'hide'} 
PROPERTY INTERNAL proCountedWarning : INT
GET
END_GET
END_PROPERTY

PROPERTY proCountedHours : UDINT
GET
END_GET
END_PROPERTY

PROPERTY proCountedStarts : UDINT
GET
END_GET
END_PROPERTY

PROPERTY INTERNAL proGetDI_MotorHand : BOOL
GET
END_GET
END_PROPERTY

{attribute 'hide'} 
PROPERTY proNotShowDI_MotorHand : BOOL
GET
END_GET
END_PROPERTY

PROPERTY proHandModul_ITF : CtaSysIO.ITF_IO
GET
END_GET
END_PROPERTY

PROPERTY proNotShowAI_ActualValue : BOOL
GET
END_GET
END_PROPERTY

PROPERTY proGetAI_ActualValue : REAL
GET
END_GET
END_PROPERTY

PROPERTY proActualValue_ITF : CtaSysIO.ITF_IO
GET
END_GET
END_PROPERTY

{attribute 'hide'} 
PROPERTY proNotShowDI_NoError : BOOL
GET
END_GET
END_PROPERTY

PROPERTY INTERNAL proGetDI_NoError : BOOL
GET
END_GET
END_PROPERTY

PROPERTY proNoError_ITF : CtaSysIO.ITF_IO
GET
END_GET
END_PROPERTY

{attribute 'hide'} 
PROPERTY proNotShowDI_RevisionSwitchOk : BOOL
GET
END_GET
END_PROPERTY

PROPERTY INTERNAL proGetDI_RevisionSwitchOK : BOOL
GET
END_GET
END_PROPERTY

PROPERTY proRevisionSwitch_ITF : CtaSysIO.ITF_IO
GET
END_GET
END_PROPERTY

{attribute 'hide'} 
PROPERTY proNotShowDI_IsOn : BOOL
GET
END_GET
END_PROPERTY

PROPERTY INTERNAL proGetDI_IsOn : BOOL
GET
END_GET
END_PROPERTY

PROPERTY proIsOn_ITF : CtaSysIO.ITF_IO
GET
END_GET
END_PROPERTY

{attribute 'hide'} 
PROPERTY proNotShowDI_MotorFuseOk : BOOL
GET
END_GET
END_PROPERTY

PROPERTY INTERNAL proGetDI_MotorFuseOk : BOOL
GET
END_GET
END_PROPERTY

PROPERTY proMotorFuse_ITF : CtaSysIO.ITF_IO
GET
END_GET
END_PROPERTY

{attribute 'hide'} 
PROPERTY proNotShowDI_FuseOk : BOOL
GET
END_GET
END_PROPERTY

PROPERTY INTERNAL proGetDI_FuseOK : BOOL
GET
END_GET
END_PROPERTY

PROPERTY proFuse_ITF : CtaSysIO.ITF_IO
GET
END_GET
END_PROPERTY

{attribute 'hide'} 
PROPERTY proNotShowDI_Ready : BOOL
GET
END_GET
END_PROPERTY

PROPERTY INTERNAL proGetDI_IsReady : BOOL
GET
END_GET
END_PROPERTY

PROPERTY proReady_ITF : CtaSysIO.ITF_IO
GET
END_GET
END_PROPERTY

PROPERTY proOn_ITF : CtaSysIO.ITF_IO
GET
END_GET
END_PROPERTY

PROPERTY proOnY_ITF : CtaSysIO.ITF_IO
GET
END_GET
END_PROPERTY

PROPERTY proIsRegulatet : BOOL
GET
END_GET
END_PROPERTY

PROPERTY proIsHandOnOrOff : BOOL
GET
END_GET
END_PROPERTY

